KUKA KRL program: MyProgram_055().src

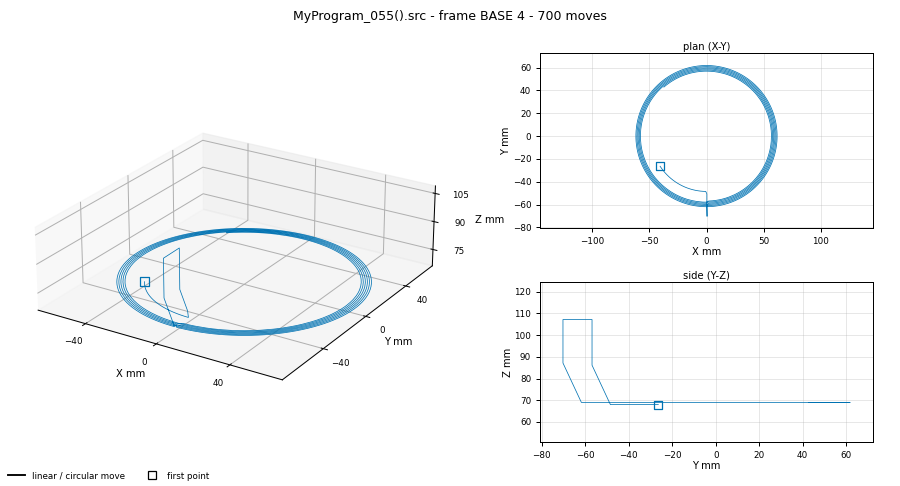
[picture p0: tool path of MyProgram_055().src in frame BASE 4, 700 of 700 moves have a stored position in this frame; points joined in program order, loops and branches not executed]
&ACCESS RVP
&REL 1
&PARAM TEMPLATE = C:\KRC\Roboter\Template\vorgabe
&PARAM EDITMASK = *
DEF MyProgram_055()
; ---- Setting reference (Base) ----
$BASE = BASE_DATA[4]

; --------------------------
; ---- Setting tool (TCP) ----
$TOOL = TOOL_DATA[3]
; --------------------------

$VEL.CP = VEL_APROX_PRINT
Startdeposition()
$VEL.CP = VEL_PRINT
LIN {X -40.6074,Y -26.4095,Z 68,A -152.5129,B 24.8688,C -2.6433,E1 24.8669,E2 236.0366} C_DIS
LIN {X -39.2547,Y -28.3812,Z 68,A -149.7049,B 24.8695,C -2.6361,E1 24.8714,E2 233.2321} C_DIS
LIN {X -37.8183,Y -30.2688,Z 68,A -146.8695,B 24.8701,C -2.63,E1 24.8763,E2 230.398} C_DIS
LIN {X -36.2912,Y -32.0839,Z 68,A -144.0489,B 24.8707,C -2.6239,E1 24.8814,E2 227.579} C_DIS
LIN {X -34.6958,Y -33.8024,Z 68,A -141.2485,B 24.8713,C -2.6184,E1 24.8868,E2 224.7796} C_DIS
LIN {X -32.9948,Y -35.4648,Z 68,A -138.4241,B 24.8718,C -2.6129,E1 24.8925,E2 221.9566} C_DIS
LIN {X -31.1918,Y -37.0607,Z 68,A -135.5745,B 24.8723,C -2.6076,E1 24.8986,E2 219.1087} C_DIS
LIN {X -29.3613,Y -38.5269,Z 68,A -132.7858,B 24.8728,C -2.6029,E1 24.9047,E2 216.3208} C_DIS
LIN {X -27.3998,Y -39.9459,Z 68,A -129.928,B 24.8733,C -2.5982,E1 24.9112,E2 213.4645} C_DIS
LIN {X -25.4106,Y -41.2399,Z 68,A -127.0866,B 24.8736,C -2.5945,E1 24.9179,E2 210.6229} C_DIS
LIN {X -23.4236,Y -42.3996,Z 68,A -124.332,B 24.8739,C -2.5914,E1 24.9246,E2 207.8677} C_DIS
LIN {X -21.2542,Y -43.5279,Z 68,A -121.4558,B 24.8743,C -2.5876,E1 24.9318,E2 204.9928} C_DIS
LIN {X -19.0978,Y -44.5162,Z 68,A -118.6602,B 24.8746,C -2.5844,E1 24.9389,E2 202.198} C_DIS
LIN {X -16.9499,Y -45.3772,Z 68,A -115.9012,B 24.8748,C -2.5823,E1 24.9461,E2 199.4383} C_DIS
LIN {X -14.6463,Y -46.1725,Z 68,A -113.0133,B 24.875,C -2.5801,E1 24.9538,E2 196.5502} C_DIS
LIN {X -12.4159,Y -46.8213,Z 68,A -110.2357,B 24.8751,C -2.5789,E1 24.9612,E2 193.7711} C_DIS
LIN {X -10.0365,Y -47.3887,Z 68,A -107.3856,B 24.8753,C -2.5768,E1 24.969,E2 190.9223} C_DIS
LIN {X -7.7033,Y -47.8234,Z 68,A -104.5763,B 24.8754,C -2.576,E1 24.9767,E2 188.1123} C_DIS
LIN {X -5.3374,Y -48.145,Z 68,A -101.7511,B 24.8754,C -2.5755,E1 24.9846,E2 185.2861} C_DIS
LIN {X -3.0451,Y -48.3437,Z 68,A -98.9821,B 24.8754,C -2.5763,E1 24.9923,E2 182.5142} C_DIS
LIN {X -0.6737,Y -48.4348,Z 68,A -96.2003,B 24.8754,C -2.5763,E1 25,E2 179.732} C_DIS
LIN {X -0.6737,Y -48.4348,Z 68,A -96.2003,B 24.8754,C -2.5763,E1 25,E2 179.732} C_DIS
Enddeposition()
LIN {X 0.3038,Y -50.5495,Z 72.5315,A -96.1445,B 24.8777,C -2.5529,E1 25,E2 179.732} C_DIS
LIN {X 0.2933,Y -56.8888,Z 86.1262,A -96.1143,B 24.8789,C -2.5402,E1 25,E2 179.732} C_DIS
LIN {X 0.2933,Y -56.8888,Z 107.1262,A -96.4674,B 24.8642,C -2.6887,E1 25,E2 179.732} C_DIS
LIN {X 0.4779,Y -70.2594,Z 107.1262,A -95.1787,B 24.8844,C -2.4821,E1 25.0023,E2 178.9343} C_DIS
LIN {X 0.4779,Y -70.2594,Z 87.1262,A -94.8425,B 24.8972,C -2.3406,E1 25.0023,E2 178.9343} C_DIS
LIN {X 0.4001,Y -63.9206,Z 73.5315,A -94.8701,B 24.8962,C -2.3523,E1 25.0023,E2 178.9343} C_DIS
LIN {X 0.3742,Y -61.8077,Z 69,A -94.8808,B 24.8958,C -2.3568,E1 25.0023,E2 178.9343} C_DIS
Startdeposition()
$VEL.CP = VEL_PRINT
LIN {X -1.5169,Y -61.7936,Z 69,A -97.6403,B 24.8977,C -2.3344,E1 24.9944,E2 181.747} C_DIS
LIN {X -4.5472,Y -61.6448,Z 69,A -100.4525,B 24.8977,C -2.3344,E1 24.9866,E2 184.5603} C_DIS
LIN {X -7.5665,Y -61.3474,Z 69,A -103.2657,B 24.8977,C -2.3346,E1 24.9788,E2 187.3745} C_DIS
LIN {X -10.5675,Y -60.9022,Z 69,A -106.0799,B 24.8977,C -2.3354,E1 24.971,E2 190.1896} C_DIS
LIN {X -13.5431,Y -60.3104,Z 69,A -108.8951,B 24.8976,C -2.3365,E1 24.9633,E2 193.0055} C_DIS
LIN {X -16.4861,Y -59.5732,Z 69,A -111.7113,B 24.8974,C -2.3381,E1 24.9557,E2 195.8221} C_DIS
LIN {X -19.3894,Y -58.6925,Z 69,A -114.5285,B 24.8973,C -2.34,E1 24.9482,E2 198.6396} C_DIS
LIN {X -22.2459,Y -57.6704,Z 69,A -117.3466,B 24.897,C -2.3424,E1 24.9408,E2 201.4578} C_DIS
LIN {X -25.0489,Y -56.5094,Z 69,A -120.1657,B 24.8968,C -2.3452,E1 24.9336,E2 204.2769} C_DIS
LIN {X -27.7915,Y -55.2122,Z 69,A -122.9858,B 24.8965,C -2.3484,E1 24.9265,E2 207.0968} C_DIS
LIN {X -30.4671,Y -53.782,Z 69,A -125.8067,B 24.8962,C -2.3519,E1 24.9196,E2 209.9173} C_DIS
LIN {X -33.0694,Y -52.2223,Z 69,A -128.6284,B 24.8959,C -2.3558,E1 24.9129,E2 212.7385} C_DIS
LIN {X -35.592,Y -50.5368,Z 69,A -131.4511,B 24.8955,C -2.3601,E1 24.9064,E2 215.5605} C_DIS
LIN {X -38.0289,Y -48.7295,Z 69,A -134.2747,B 24.8951,C -2.3648,E1 24.9001,E2 218.3832} C_DIS
LIN {X -40.3741,Y -46.8048,Z 69,A -137.0991,B 24.8946,C -2.3698,E1 24.8941,E2 221.2065} C_DIS
LIN {X -42.6125,Y -44.7764,Z 69,A -139.915,B 24.8942,C -2.375,E1 24.8883,E2 224.0214} C_DIS
LIN {X -44.7673,Y -42.6221,Z 69,A -142.7502,B 24.8936,C -2.3807,E1 24.8828,E2 226.8551} C_DIS
LIN {X -46.8048,Y -40.3741,Z 69,A -145.5768,B 24.8931,C -2.3867,E1 24.8776,E2 229.6802} C_DIS
LIN {X -48.7295,Y -38.0289,Z 69,A -148.4042,B 24.8925,C -2.393,E1 24.8727,E2 232.5058} C_DIS
LIN {X -50.5368,Y -35.592,Z 69,A -151.2322,B 24.892,C -2.3995,E1 24.868,E2 235.332} C_DIS
LIN {X -52.2223,Y -33.0694,Z 69,A -154.0608,B 24.8913,C -2.4063,E1 24.8637,E2 238.1586} C_DIS
LIN {X -53.782,Y -30.4671,Z 69,A -156.8901,B 24.8907,C -2.4133,E1 24.8597,E2 240.9858} C_DIS
LIN {X -55.2122,Y -27.7915,Z 69,A -159.7199,B 24.89,C -2.4206,E1 24.8561,E2 243.8133} C_DIS
LIN {X -56.5094,Y -25.0489,Z 69,A -162.5501,B 24.8894,C -2.4281,E1 24.8528,E2 246.6411} C_DIS
LIN {X -57.6704,Y -22.2459,Z 69,A -165.3808,B 24.8887,C -2.4357,E1 24.8499,E2 249.4694} C_DIS
LIN {X -58.6925,Y -19.3894,Z 69,A -168.212,B 24.8879,C -2.4436,E1 24.8473,E2 252.298} C_DIS
LIN {X -59.5732,Y -16.4861,Z 69,A -171.0435,B 24.8872,C -2.4516,E1 24.8451,E2 255.1266} C_DIS
LIN {X -60.3104,Y -13.5431,Z 69,A -173.8753,B 24.8864,C -2.4597,E1 24.8433,E2 257.9557} C_DIS
LIN {X -60.9022,Y -10.5675,Z 69,A -176.7075,B 24.8857,C -2.468,E1 24.8418,E2 260.7849} C_DIS
LIN {X -61.3474,Y -7.5665,Z 69,A -179.5398,B 24.8849,C -2.4763,E1 24.8408,E2 263.6142} C_DIS
LIN {X -61.6448,Y -4.5472,Z 69,A 177.6277,B 24.8841,C -2.4847,E1 24.8401,E2 266.4436} C_DIS
LIN {X -61.7936,Y -1.5169,Z 69,A 174.8866,B 24.8832,C -2.4949,E1 24.8398,E2 269.177} C_DIS
LIN {X -61.7936,Y 1.5169,Z 69,A 171.9622,B 24.8825,C -2.5017,E1 24.8398,E2 272.1025} C_DIS
LIN {X -61.6448,Y 4.5472,Z 69,A 169.1296,B 24.8817,C -2.5102,E1 24.8404,E2 274.9319} C_DIS
LIN {X -61.3474,Y 7.5665,Z 69,A 166.2969,B 24.8809,C -2.5188,E1 24.8412,E2 277.7612} C_DIS
LIN {X -60.9022,Y 10.5675,Z 69,A 163.4642,B 24.8801,C -2.5272,E1 24.8425,E2 280.5904} C_DIS
LIN {X -60.3104,Y 13.5431,Z 69,A 160.6317,B 24.8793,C -2.5357,E1 24.8441,E2 283.4195} C_DIS
LIN {X -59.5732,Y 16.4861,Z 69,A 157.7993,B 24.8785,C -2.544,E1 24.8461,E2 286.2484} C_DIS
LIN {X -58.6925,Y 19.3894,Z 69,A 154.9672,B 24.8777,C -2.5523,E1 24.8485,E2 289.077} C_DIS
LIN {X -57.6704,Y 22.2459,Z 69,A 152.1353,B 24.8769,C -2.5605,E1 24.8513,E2 291.9053} C_DIS
LIN {X -56.5094,Y 25.0489,Z 69,A 149.3037,B 24.8761,C -2.5685,E1 24.8544,E2 294.7334} C_DIS
LIN {X -55.2122,Y 27.7915,Z 69,A 146.4725,B 24.8754,C -2.5763,E1 24.8578,E2 297.5612} C_DIS
LIN {X -53.782,Y 30.4671,Z 69,A 143.6416,B 24.8746,C -2.584,E1 24.8616,E2 300.3885} C_DIS
LIN {X -52.2223,Y 33.0694,Z 69,A 140.8113,B 24.8739,C -2.5916,E1 24.8658,E2 303.2154} C_DIS
LIN {X -50.5368,Y 35.592,Z 69,A 137.9814,B 24.8732,C -2.5989,E1 24.8702,E2 306.0419} C_DIS
LIN {X -48.7295,Y 38.0289,Z 69,A 135.1522,B 24.8725,C -2.606,E1 24.875,E2 308.8677} C_DIS
LIN {X -46.8048,Y 40.3741,Z 69,A 132.3234,B 24.8718,C -2.6128,E1 24.8801,E2 311.6931} C_DIS
LIN {X -44.7673,Y 42.6221,Z 69,A 129.4952,B 24.8712,C -2.6194,E1 24.8855,E2 314.518} C_DIS
LIN {X -42.6221,Y 44.7673,Z 69,A 126.6678,B 24.8706,C -2.6257,E1 24.8911,E2 317.3422} C_DIS
LIN {X -40.3741,Y 46.8048,Z 69,A 123.8408,B 24.87,C -2.6317,E1 24.897,E2 320.166} C_DIS
LIN {X -38.0289,Y 48.7295,Z 69,A 121.0148,B 24.8694,C -2.6374,E1 24.9032,E2 322.9889} C_DIS
LIN {X -35.592,Y 50.5368,Z 69,A 118.1895,B 24.8689,C -2.6428,E1 24.9095,E2 325.8113} C_DIS
LIN {X -33.0694,Y 52.2223,Z 69,A 115.365,B 24.8683,C -2.6479,E1 24.9161,E2 328.6328} C_DIS
LIN {X -30.4671,Y 53.782,Z 69,A 112.5412,B 24.8679,C -2.6526,E1 24.9229,E2 331.4539} C_DIS
LIN {X -27.8247,Y 55.1952,Z 69,A 109.7441,B 24.8675,C -2.6567,E1 24.9299,E2 334.2487} C_DIS
LIN {X -25.0489,Y 56.5094,Z 69,A 106.8964,B 24.867,C -2.661,E1 24.9371,E2 337.0934} C_DIS
LIN {X -22.2459,Y 57.6704,Z 69,A 104.0752,B 24.8667,C -2.6646,E1 24.9444,E2 339.9121} C_DIS
LIN {X -19.3894,Y 58.6925,Z 69,A 101.2549,B 24.8663,C -2.6678,E1 24.9518,E2 342.7301} C_DIS
LIN {X -16.4861,Y 59.5732,Z 69,A 98.4357,B 24.8661,C -2.6707,E1 24.9594,E2 345.5471} C_DIS
LIN {X -13.5431,Y 60.3104,Z 69,A 95.6173,B 24.8658,C -2.6731,E1 24.967,E2 348.3634} C_DIS
LIN {X -10.5675,Y 60.9022,Z 69,A 92.7999,B 24.8656,C -2.6752,E1 24.9748,E2 351.179} C_DIS
LIN {X -7.6019,Y 61.3428,Z 69,A 90.0082,B 24.8655,C -2.6767,E1 24.9825,E2 353.9694} C_DIS
LIN {X -4.5472,Y 61.6448,Z 69,A 87.168,B 24.8653,C -2.6781,E1 24.9904,E2 356.8075} C_DIS
LIN {X -1.5169,Y 61.7936,Z 69,A 84.3535,B 24.8653,C -2.6789,E1 24.9982,E2 359.6205} C_DIS
LIN {X 1.5169,Y 61.7936,Z 69,A 81.54,B 24.8652,C -2.6793,E1 25.0061,E2 362.4328} C_DIS
LIN {X 4.5472,Y 61.6448,Z 69,A 78.7275,B 24.8652,C -2.6793,E1 25.0139,E2 365.244} C_DIS
LIN {X 7.5665,Y 61.3474,Z 69,A 75.9161,B 24.8652,C -2.6789,E1 25.0217,E2 368.0545} C_DIS
LIN {X 10.5675,Y 60.9022,Z 69,A 73.1055,B 24.8653,C -2.6781,E1 25.0295,E2 370.8643} C_DIS
LIN {X 13.5431,Y 60.3104,Z 69,A 70.296,B 24.8654,C -2.6769,E1 25.0371,E2 373.6732} C_DIS
LIN {X 16.4861,Y 59.5732,Z 69,A 67.4874,B 24.8656,C -2.6752,E1 25.0447,E2 376.4812} C_DIS
LIN {X 19.3894,Y 58.6925,Z 69,A 64.6798,B 24.8658,C -2.6732,E1 25.0522,E2 379.2886} C_DIS
LIN {X 22.2459,Y 57.6704,Z 69,A 61.8732,B 24.8661,C -2.6707,E1 25.0596,E2 382.0951} C_DIS
LIN {X 25.0489,Y 56.5094,Z 69,A 59.0674,B 24.8663,C -2.6679,E1 25.0668,E2 384.9009} C_DIS
LIN {X 27.7915,Y 55.2122,Z 69,A 56.2625,B 24.8667,C -2.6646,E1 25.0738,E2 387.706} C_DIS
LIN {X 30.4671,Y 53.782,Z 69,A 53.4587,B 24.867,C -2.661,E1 25.0807,E2 390.5102} C_DIS
LIN {X 33.0694,Y 52.2223,Z 69,A 50.6555,B 24.8674,C -2.6571,E1 25.0873,E2 393.314} C_DIS
LIN {X 35.592,Y 50.5368,Z 69,A 47.8533,B 24.8679,C -2.6528,E1 25.0938,E2 396.1169} C_DIS
LIN {X 38.0289,Y 48.7295,Z 69,A 45.0519,B 24.8683,C -2.6481,E1 25.1,E2 398.9192} C_DIS
LIN {X 40.3741,Y 46.8048,Z 69,A 42.2512,B 24.8688,C -2.6431,E1 25.106,E2 401.7209} C_DIS
LIN {X 42.6221,Y 44.7673,Z 69,A 39.4515,B 24.8694,C -2.6377,E1 25.1117,E2 404.5219} C_DIS
LIN {X 44.7673,Y 42.6221,Z 69,A 36.6525,B 24.8699,C -2.6321,E1 25.1172,E2 407.3223} C_DIS
LIN {X 46.8048,Y 40.3741,Z 69,A 33.8542,B 24.8705,C -2.6261,E1 25.1224,E2 410.1222} C_DIS
LIN {X 48.7295,Y 38.0289,Z 69,A 31.0563,B 24.8711,C -2.6199,E1 25.1273,E2 412.9217} C_DIS
LIN {X 50.5368,Y 35.592,Z 69,A 28.2593,B 24.8718,C -2.6134,E1 25.1318,E2 415.7205} C_DIS
LIN {X 52.2223,Y 33.0694,Z 69,A 25.4629,B 24.8724,C -2.6067,E1 25.1361,E2 418.5189} C_DIS
LIN {X 53.782,Y 30.4671,Z 69,A 22.667,B 24.8731,C -2.5997,E1 25.14,E2 421.3169} C_DIS
LIN {X 55.2122,Y 27.7915,Z 69,A 19.8717,B 24.8738,C -2.5925,E1 25.1436,E2 424.1145} C_DIS
LIN {X 56.5094,Y 25.0489,Z 69,A 17.0768,B 24.8745,C -2.5851,E1 25.1469,E2 426.9117} C_DIS
LIN {X 57.6704,Y 22.2459,Z 69,A 14.2823,B 24.8753,C -2.5775,E1 25.1498,E2 429.7087} C_DIS
LIN {X 58.6925,Y 19.3894,Z 69,A 11.4883,B 24.876,C -2.5697,E1 25.1523,E2 432.5054} C_DIS
LIN {X 59.5732,Y 16.4861,Z 69,A 8.6946,B 24.8768,C -2.5618,E1 25.1545,E2 435.3019} C_DIS
LIN {X 60.3104,Y 13.5431,Z 69,A 5.9012,B 24.8776,C -2.5537,E1 25.1563,E2 438.098} C_DIS
LIN {X 60.9022,Y 10.5675,Z 69,A 3.1081,B 24.8784,C -2.5456,E1 25.1578,E2 440.8941} C_DIS
LIN {X 61.3474,Y 7.5665,Z 69,A 0.3152,B 24.8791,C -2.5373,E1 25.1588,E2 443.6901} C_DIS
LIN {X 61.6448,Y 4.5472,Z 69,A -2.4776,B 24.8799,C -2.529,E1 25.1595,E2 446.4859} C_DIS
LIN {X 61.7936,Y 1.5169,Z 69,A -5.18,B 24.8805,C -2.5229,E1 25.1598,E2 449.1868} C_DIS
LIN {X 61.7936,Y -1.5169,Z 69,A -8.0628,B 24.8815,C -2.5122,E1 25.1597,E2 452.0775} C_DIS
LIN {X 61.6448,Y -4.5472,Z 69,A -10.8552,B 24.8823,C -2.5038,E1 25.1592,E2 454.8732} C_DIS
LIN {X 61.3474,Y -7.5665,Z 69,A -13.6477,B 24.8831,C -2.4954,E1 25.1583,E2 457.6691} C_DIS
LIN {X 60.9022,Y -10.5675,Z 69,A -16.4402,B 24.8839,C -2.487,E1 25.1571,E2 460.4651} C_DIS
LIN {X 60.3104,Y -13.5431,Z 69,A -19.2329,B 24.8847,C -2.4787,E1 25.1555,E2 463.2612} C_DIS
LIN {X 59.5732,Y -16.4861,Z 69,A -22.0257,B 24.8855,C -2.4704,E1 25.1535,E2 466.0575} C_DIS
LIN {X 58.6925,Y -19.3894,Z 69,A -24.8188,B 24.8862,C -2.4622,E1 25.1511,E2 468.854} C_DIS
LIN {X 57.6704,Y -22.2459,Z 69,A -27.612,B 24.887,C -2.4542,E1 25.1484,E2 471.6507} C_DIS
LIN {X 56.5094,Y -25.0489,Z 69,A -30.4057,B 24.8877,C -2.4462,E1 25.1454,E2 474.4479} C_DIS
LIN {X 55.2122,Y -27.7915,Z 69,A -33.1997,B 24.8884,C -2.4384,E1 25.1419,E2 477.2454} C_DIS
LIN {X 53.782,Y -30.4671,Z 69,A -35.994,B 24.8891,C -2.4307,E1 25.1382,E2 480.0432} C_DIS
LIN {X 52.2223,Y -33.0694,Z 69,A -38.7886,B 24.8898,C -2.4233,E1 25.1341,E2 482.8413} C_DIS
LIN {X 50.5368,Y -35.592,Z 69,A -41.5839,B 24.8905,C -2.416,E1 25.1296,E2 485.6399} C_DIS
LIN {X 48.7295,Y -38.0289,Z 69,A -44.3797,B 24.8911,C -2.4089,E1 25.1249,E2 488.4391} C_DIS
LIN {X 46.8048,Y -40.3741,Z 69,A -47.1759,B 24.8917,C -2.4021,E1 25.1199,E2 491.2387} C_DIS
LIN {X 44.7673,Y -42.6221,Z 69,A -49.9729,B 24.8923,C -2.3955,E1 25.1146,E2 494.039} C_DIS
LIN {X 42.6221,Y -44.7673,Z 69,A -52.7703,B 24.8929,C -2.3892,E1 25.109,E2 496.8396} C_DIS
LIN {X 40.3741,Y -46.8048,Z 69,A -55.5685,B 24.8934,C -2.3832,E1 25.1031,E2 499.641} C_DIS
LIN {X 38.0289,Y -48.7295,Z 69,A -58.3673,B 24.8939,C -2.3775,E1 25.097,E2 502.4429} C_DIS
LIN {X 35.592,Y -50.5368,Z 69,A -61.1669,B 24.8944,C -2.372,E1 25.0907,E2 505.2455} C_DIS
LIN {X 33.0694,Y -52.2223,Z 69,A -63.9673,B 24.8949,C -2.3669,E1 25.0841,E2 508.0487} C_DIS
LIN {X 30.4671,Y -53.782,Z 69,A -66.7685,B 24.8953,C -2.3622,E1 25.0773,E2 510.8528} C_DIS
LIN {X 27.7915,Y -55.2122,Z 69,A -69.5705,B 24.8957,C -2.3577,E1 25.0704,E2 513.6574} C_DIS
LIN {X 25.0489,Y -56.5094,Z 69,A -72.3733,B 24.8961,C -2.3537,E1 25.0633,E2 516.4628} C_DIS
LIN {X 22.2459,Y -57.6704,Z 69,A -75.177,B 24.8964,C -2.35,E1 25.056,E2 519.269} C_DIS
LIN {X 19.3894,Y -58.6925,Z 69,A -77.9817,B 24.8967,C -2.3466,E1 25.0486,E2 522.076} C_DIS
LIN {X 16.4861,Y -59.5732,Z 69,A -80.7871,B 24.8969,C -2.3437,E1 25.0411,E2 524.8836} C_DIS
LIN {X 13.5431,Y -60.3104,Z 69,A -83.5936,B 24.8972,C -2.3411,E1 25.0334,E2 527.6921} C_DIS
LIN {X 10.5675,Y -60.9022,Z 69,A -86.401,B 24.8973,C -2.339,E1 25.0257,E2 530.5015} C_DIS
LIN {X 7.5665,Y -61.3474,Z 69,A -89.2093,B 24.8975,C -2.3372,E1 25.0179,E2 533.3116} C_DIS
LIN {X 4.5472,Y -61.6448,Z 69,A -92.0187,B 24.8976,C -2.3359,E1 25.0101,E2 536.1226} C_DIS
LIN {X 1.5169,Y -61.7936,Z 69,A -94.829,B 24.8977,C -2.335,E1 25.0023,E2 538.9343} C_DIS
LIN {X 1.5169,Y -61.7936,Z 69,A -94.829,B 24.8977,C -2.335,E1 25.0023,E2 538.9343} C_DIS
Enddeposition()
LIN {X 0.3699,Y -60.8218,Z 69,A -95.3511,B 24.8952,C -2.3637,E1 25.001,E2 539.3882} C_DIS
Startdeposition()
$VEL.CP = VEL_PRINT
LIN {X 3.5241,Y -60.721,Z 69,A -91.7282,B 24.8938,C -2.3788,E1 25.0112,E2 535.7302} C_DIS
LIN {X 6.9367,Y -60.4263,Z 69,A -88.4115,B 24.8935,C -2.3825,E1 25.0205,E2 532.4068} C_DIS
LIN {X 9.7316,Y -60.0402,Z 69,A -84.8923,B 24.8916,C -2.4038,E1 25.0303,E2 528.8406} C_DIS
LIN {X 13.0357,Y -59.4097,Z 69,A -82.7107,B 24.8933,C -2.3843,E1 25.0361,E2 526.7081} C_DIS
LIN {X 15.5224,Y -58.81,Z 69,A -80.1105,B 24.8927,C -2.391,E1 25.0432,E2 524.0959} C_DIS
LIN {X 17.6784,Y -58.1982,Z 69,A -78.3032,B 24.8931,C -2.3864,E1 25.048,E2 522.3025} C_DIS
LIN {X 20.9532,Y -57.1,Z 69,A -74.8965,B 24.8925,C -2.394,E1 25.057,E2 518.8847} C_DIS
LIN {X 23.4984,Y -56.1006,Z 69,A -72.2344,B 24.8919,C -2.3996,E1 25.0639,E2 516.2154} C_DIS
LIN {X 26.0446,Y -54.9656,Z 69,A -68.804,B 24.8899,C -2.4224,E1 25.0727,E2 512.7398} C_DIS
LIN {X 29.0105,Y -53.4586,Z 69,A -66.3744,B 24.8909,C -2.4112,E1 25.0786,E2 510.3437} C_DIS
LIN {X 31.8828,Y -51.798,Z 69,A -63.3879,B 24.8907,C -2.4135,E1 25.0857,E2 507.3608} C_DIS
LIN {X 34.4186,Y -50.1491,Z 69,A -60.7942,B 24.8907,C -2.4131,E1 25.0917,E2 504.7769} C_DIS
LIN {X 37.3365,Y -48.0155,Z 69,A -57.1659,B 24.8896,C -2.4254,E1 25.0999,E2 501.1324} C_DIS
LIN {X 39.6383,Y -46.1336,Z 69,A -54.7199,B 24.8898,C -2.4231,E1 25.1051,E2 498.7012} C_DIS
LIN {X 41.8601,Y -44.1275,Z 69,A -51.5668,B 24.8885,C -2.4376,E1 25.1116,E2 495.5267} C_DIS
LIN {X 44.7982,Y -41.1407,Z 69,A -47.6443,B 24.8877,C -2.4466,E1 25.1192,E2 491.5998} C_DIS
LIN {X 46.9752,Y -38.6376,Z 69,A -44.2528,B 24.8863,C -2.461,E1 25.1254,E2 488.1896} C_DIS
LIN {X 49.0255,Y -35.9992,Z 69,A -41.6748,B 24.8868,C -2.4556,E1 25.1297,E2 485.6369} C_DIS
LIN {X 50.7232,Y -33.565,Z 69,A -38.4521,B 24.8852,C -2.4736,E1 25.1348,E2 482.3874} C_DIS
LIN {X 52.2264,Y -31.1755,Z 69,A -35.773,B 24.8844,C -2.4816,E1 25.1386,E2 479.7031} C_DIS
LIN {X 53.8881,Y -28.2053,Z 69,A -32.8097,B 24.8841,C -2.4849,E1 25.1426,E2 476.7475} C_DIS
LIN {X 55.2151,Y -25.5099,Z 69,A -30.0221,B 24.8834,C -2.4922,E1 25.1459,E2 473.9577} C_DIS
LIN {X 56.1602,Y -23.3571,Z 69,A -27.557,B 24.8822,C -2.505,E1 25.1486,E2 471.476} C_DIS
LIN {X 57.3545,Y -20.2464,Z 69,A -24.8024,B 24.8822,C -2.505,E1 25.1513,E2 468.7365} C_DIS
LIN {X 58.0728,Y -18.083,Z 69,A -22.7658,B 24.8818,C -2.5089,E1 25.153,E2 466.7024} C_DIS
LIN {X 58.8136,Y -15.5078,Z 69,A -20.0069,B 24.8806,C -2.5225,E1 25.155,E2 463.9271} C_DIS
LIN {X 59.6377,Y -11.9522,Z 69,A -16.6322,B 24.8797,C -2.5317,E1 25.1571,E2 460.5503} C_DIS
LIN {X 60.0812,Y -9.4722,Z 69,A -13.8457,B 24.878,C -2.5495,E1 25.1583,E2 457.7383} C_DIS
LIN {X 60.5662,Y -5.5828,Z 69,A -10.6448,B 24.878,C -2.5489,E1 25.1593,E2 454.5575} C_DIS
LIN {X 60.7566,Y -2.8512,Z 69,A -8.1375,B 24.8774,C -2.5553,E1 25.1597,E2 452.05} C_DIS
LIN {X 60.8244,Y -0.2246,Z 69,A -5.502,B 24.8763,C -2.5671,E1 25.1597,E2 449.4025} C_DIS
LIN {X 60.7088,Y 3.7418,Z 69,A -1.8226,B 24.8753,C -2.5774,E1 25.1593,E2 445.7205} C_DIS
LIN {X 60.3426,Y 7.6319,Z 69,A 1.9824,B 24.8739,C -2.5919,E1 25.1582,E2 441.9037} C_DIS
LIN {X 59.8211,Y 10.9965,Z 69,A 5.4528,B 24.8723,C -2.6083,E1 25.1565,E2 438.4149} C_DIS
LIN {X 58.6681,Y 16.0475,Z 69,A 9.7585,B 24.8723,C -2.6088,E1 25.1536,E2 434.1328} C_DIS
LIN {X 57.8754,Y 18.705,Z 69,A 12.3693,B 24.8715,C -2.6165,E1 25.1515,E2 431.5186} C_DIS
LIN {X 56.9734,Y 21.2964,Z 69,A 14.8842,B 24.8709,C -2.6223,E1 25.1491,E2 429.0041} C_DIS
LIN {X 55.9024,Y 23.9686,Z 69,A 17.7553,B 24.8697,C -2.6339,E1 25.146,E2 426.1216} C_DIS
LIN {X 54.968,Y 26.0397,Z 69,A 19.8777,B 24.8692,C -2.6393,E1 25.1435,E2 423.9977} C_DIS
LIN {X 53.6349,Y 28.6855,Z 69,A 22.5302,B 24.8688,C -2.6436,E1 25.1401,E2 421.3492} C_DIS
LIN {X 52.3266,Y 31.0059,Z 69,A 25.1098,B 24.868,C -2.6519,E1 25.1365,E2 418.7633} C_DIS
LIN {X 51.0461,Y 33.0727,Z 69,A 27.3319,B 24.8675,C -2.6561,E1 25.1331,E2 416.5424} C_DIS
LIN {X 49.5259,Y 35.3075,Z 69,A 29.8988,B 24.8668,C -2.6628,E1 25.129,E2 413.972} C_DIS
LIN {X 47.6836,Y 37.7586,Z 69,A 32.4782,B 24.8668,C -2.6624,E1 25.1246,E2 411.406} C_DIS
LIN {X 44.7969,Y 41.1421,Z 69,A 37.0286,B 24.8651,C -2.6803,E1 25.1163,E2 406.8337} C_DIS
LIN {X 42.4394,Y 43.5711,Z 69,A 39.7141,B 24.8656,C -2.6752,E1 25.111,E2 404.1717} C_DIS
LIN {X 39.5796,Y 46.1836,Z 69,A 43.7208,B 24.864,C -2.6906,E1 25.1027,E2 400.1445} C_DIS
LIN {X 37.4821,Y 47.9022,Z 69,A 46.1859,B 24.8638,C -2.6932,E1 25.0973,E2 397.6825} C_DIS
LIN {X 35.4881,Y 49.3971,Z 69,A 48.479,B 24.8635,C -2.6959,E1 25.0921,E2 395.3911} C_DIS
LIN {X 33.2095,Y 50.9575,Z 69,A 50.9932,B 24.8633,C -2.6981,E1 25.0863,E2 392.8802} C_DIS
LIN {X 31.29,Y 52.1582,Z 69,A 53.1478,B 24.8629,C -2.7017,E1 25.0812,E2 390.7237} C_DIS
LIN {X 29.1742,Y 53.3699,Z 69,A 55.6356,B 24.8622,C -2.7092,E1 25.0751,E2 388.2256} C_DIS
LIN {X 26.4475,Y 54.7721,Z 69,A 58.483,B 24.8619,C -2.7118,E1 25.068,E2 385.3796} C_DIS
LIN {X 23.9448,Y 55.9125,Z 69,A 61.1419,B 24.8614,C -2.7162,E1 25.0612,E2 382.7169} C_DIS
LIN {X 21.3004,Y 56.9719,Z 69,A 63.7978,B 24.8612,C -2.7181,E1 25.0542,E2 380.0621} C_DIS
LIN {X 18.5844,Y 57.9144,Z 69,A 66.505,B 24.861,C -2.7203,E1 25.0471,E2 377.3549} C_DIS
LIN {X 16.1062,Y 58.6523,Z 69,A 69.0598,B 24.8606,C -2.7245,E1 25.0402,E2 374.7944} C_DIS
LIN {X 12.5567,Y 59.5137,Z 69,A 72.275,B 24.8609,C -2.7213,E1 25.0315,E2 371.591} C_DIS
LIN {X 9.9654,Y 60.0011,Z 69,A 74.4475,B 24.8615,C -2.7156,E1 25.0255,E2 369.4347} C_DIS
LIN {X 7.7997,Y 60.3208,Z 69,A 78.057,B 24.858,C -2.7494,E1 25.0153,E2 365.7477} C_DIS
LIN {X 3.6725,Y 60.7128,Z 69,A 80.3983,B 24.8615,C -2.716,E1 25.009,E2 363.4869} C_DIS
LIN {X -0.0244,Y 60.824,Z 69,A 84.239,B 24.8607,C -2.723,E1 24.9983,E2 359.6301} C_DIS
LIN {X -2.9809,Y 60.751,Z 69,A 86.9887,B 24.8609,C -2.7214,E1 24.9906,E2 356.8837} C_DIS
LIN {X -5.8016,Y 60.546,Z 69,A 89.7033,B 24.8609,C -2.7213,E1 24.983,E2 354.1683} C_DIS
LIN {X -10.4137,Y 59.9255,Z 69,A 94.0806,B 24.8612,C -2.7182,E1 24.971,E2 349.7945} C_DIS
LIN {X -13.7016,Y 59.2596,Z 69,A 97.2928,B 24.8614,C -2.7166,E1 24.9622,E2 346.5823} C_DIS
LIN {X -16.4479,Y 58.557,Z 69,A 99.9665,B 24.8617,C -2.714,E1 24.955,E2 343.9107} C_DIS
LIN {X -19.0418,Y 57.7663,Z 69,A 102.4277,B 24.8622,C -2.7092,E1 24.9485,E2 341.4566} C_DIS
LIN {X -23.2617,Y 56.1995,Z 69,A 106.3977,B 24.8633,C -2.6983,E1 24.9382,E2 337.5041} C_DIS
LIN {X -26.378,Y 54.8054,Z 69,A 109.7592,B 24.8635,C -2.6964,E1 24.9296,E2 334.139} C_DIS
LIN {X -27.9233,Y 54.0352,Z 69,A 112.467,B 24.8616,C -2.715,E1 24.9228,E2 331.3795} C_DIS
LIN {X -30.8335,Y 52.4285,Z 69,A 114.7128,B 24.8639,C -2.6922,E1 24.9175,E2 329.1814} C_DIS
LIN {X -33.2267,Y 50.9462,Z 69,A 117.3953,B 24.8643,C -2.6878,E1 24.9111,E2 326.5007} C_DIS
LIN {X -35.6247,Y 49.2996,Z 69,A 120.2042,B 24.8647,C -2.6837,E1 24.9047,E2 323.6919} C_DIS
LIN {X -38.0459,Y 47.4557,Z 69,A 123.3465,B 24.8648,C -2.683,E1 24.8978,E2 320.5398} C_DIS
LIN {X -41.0603,Y 44.872,Z 69,A 126.7217,B 24.8664,C -2.6677,E1 24.8908,E2 317.1877} C_DIS
LIN {X -43.1122,Y 42.9049,Z 69,A 129.5063,B 24.8668,C -2.6634,E1 24.8852,E2 314.4016} C_DIS
LIN {X -45.1474,Y 40.7579,Z 69,A 131.8856,B 24.8682,C -2.649,E1 24.8807,E2 312.0463} C_DIS
LIN {X -46.6661,Y 39.0096,Z 69,A 135.0862,B 24.8669,C -2.6625,E1 24.8749,E2 308.7988} C_DIS
LIN {X -49.2279,Y 35.7228,Z 69,A 138.4377,B 24.869,C -2.6414,E1 24.8693,E2 305.4817} C_DIS
LIN {X -50.7628,Y 33.5048,Z 69,A 141.0102,B 24.8696,C -2.6351,E1 24.8653,E2 302.9115} C_DIS
LIN {X -52.0957,Y 31.3931,Z 69,A 143.9984,B 24.8691,C -2.6403,E1 24.861,E2 299.8955} C_DIS
LIN {X -54.1446,Y 27.7093,Z 69,A 147.3916,B 24.8713,C -2.6182,E1 24.8565,E2 296.5371} C_DIS
LIN {X -55.184,Y 25.5767,Z 69,A 149.7296,B 24.8718,C -2.6135,E1 24.8538,E2 294.1975} C_DIS
LIN {X -56.4618,Y 22.619,Z 69,A 152.6761,B 24.8728,C -2.6028,E1 24.8506,E2 291.2603} C_DIS
LIN {X -57.4388,Y 20.0061,Z 69,A 155.3015,B 24.8736,C -2.5948,E1 24.8481,E2 288.6391} C_DIS
LIN {X -58.2751,Y 17.4201,Z 69,A 157.8501,B 24.8744,C -2.5868,E1 24.846,E2 286.0952} C_DIS
LIN {X -59.0128,Y 14.7319,Z 69,A 160.1902,B 24.8757,C -2.5735,E1 24.8444,E2 283.7732} C_DIS
LIN {X -59.433,Y 12.9288,Z 69,A 162.2542,B 24.8757,C -2.5738,E1 24.8431,E2 281.6962} C_DIS
LIN {X -59.964,Y 10.1871,Z 69,A 164.8902,B 24.8764,C -2.5656,E1 24.8418,E2 279.0641} C_DIS
LIN {X -60.3844,Y 7.2944,Z 69,A 167.7265,B 24.8771,C -2.5584,E1 24.8407,E2 276.2282} C_DIS
LIN {X -60.6651,Y 4.379,Z 69,A 170.6353,B 24.8777,C -2.5524,E1 24.84,E2 273.3162} C_DIS
LIN {X -60.7919,Y 1.9468,Z 69,A 172.5622,B 24.879,C -2.5386,E1 24.8398,E2 271.4109} C_DIS
LIN {X -60.8219,Y -0.493,Z 69,A 175.2013,B 24.8791,C -2.5374,E1 24.8398,E2 268.7585} C_DIS
LIN {X -60.7323,Y -3.3196,Z 69,A 177.8663,B 24.8799,C -2.5291,E1 24.8401,E2 266.0974} C_DIS
LIN {X -60.5142,Y -6.1249,Z 69,A -179.6063,B 24.8809,C -2.5186,E1 24.8408,E2 263.5799} C_DIS
LIN {X -60.1684,Y -8.9064,Z 69,A -176.772,B 24.8814,C -2.5139,E1 24.8419,E2 260.7399} C_DIS
LIN {X -59.6262,Y -12.0083,Z 69,A -173.9619,B 24.8825,C -2.502,E1 24.8433,E2 257.9417} C_DIS
LIN {X -59.0014,Y -14.7785,Z 69,A -171.3606,B 24.8834,C -2.4926,E1 24.845,E2 255.3476} C_DIS
LIN {X -58.5565,Y -16.4495,Z 69,A -169.5667,B 24.8836,C -2.4908,E1 24.8463,E2 253.5477} C_DIS
LIN {X -57.7201,Y -19.1807,Z 69,A -166.836,B 24.8842,C -2.4836,E1 24.8486,E2 250.8185} C_DIS
LIN {X -56.7436,Y -21.9028,Z 69,A -164.0819,B 24.8849,C -2.4763,E1 24.8513,E2 248.0663} C_DIS
LIN {X -54.6571,Y -26.6865,Z 69,A -158.7948,B 24.8855,C -2.4695,E1 24.8574,E2 242.7665} C_DIS
LIN {X -52.9066,Y -30.0074,Z 69,A -155.8669,B 24.8875,C -2.4487,E1 24.8613,E2 239.8728} C_DIS
LIN {X -51.7465,Y -31.9661,Z 69,A -153.4161,B 24.8875,C -2.4489,E1 24.8648,E2 237.409} C_DIS
LIN {X -50.2012,Y -34.3418,Z 69,A -150.7503,B 24.8881,C -2.4421,E1 24.869,E2 234.746} C_DIS
LIN {X -48.6003,Y -36.5712,Z 69,A -148.1528,B 24.8886,C -2.4361,E1 24.8733,E2 232.1502} C_DIS
LIN {X -46.7849,Y -38.8665,Z 69,A -145.4654,B 24.8893,C -2.4284,E1 24.878,E2 229.4687} C_DIS
LIN {X -45.1324,Y -40.7747,Z 69,A -142.9432,B 24.8896,C -2.4259,E1 24.8827,E2 226.9412} C_DIS
LIN {X -43.0487,Y -42.9691,Z 69,A -140.1657,B 24.8902,C -2.4185,E1 24.888,E2 224.1695} C_DIS
LIN {X -41.0534,Y -44.8783,Z 69,A -137.4786,B 24.8905,C -2.415,E1 24.8935,E2 221.4797} C_DIS
LIN {X -38.8702,Y -46.7818,Z 69,A -134.7466,B 24.891,C -2.4099,E1 24.8993,E2 218.7491} C_DIS
LIN {X -36.6016,Y -48.5774,Z 69,A -132.1771,B 24.8917,C -2.4021,E1 24.905,E2 216.189} C_DIS
LIN {X -34.4272,Y -50.143,Z 69,A -129.4656,B 24.8917,C -2.4017,E1 24.9112,E2 213.4692} C_DIS
LIN {X -31.6078,Y -51.9652,Z 69,A -126.3568,B 24.8923,C -2.3959,E1 24.9185,E2 210.3643} C_DIS
LIN {X -29.293,Y -53.3054,Z 69,A -123.6738,B 24.8923,C -2.3958,E1 24.9251,E2 207.6738} C_DIS
LIN {X -26.6861,Y -54.6573,Z 69,A -120.9521,B 24.8927,C -2.3915,E1 24.9319,E2 204.955} C_DIS
LIN {X -23.8336,Y -55.9593,Z 69,A -118.1485,B 24.8932,C -2.3853,E1 24.939,E2 202.1595} C_DIS
LIN {X -21.8065,Y -56.7802,Z 69,A -115.8965,B 24.8931,C -2.3873,E1 24.9449,E2 199.8979} C_DIS
LIN {X -19.3373,Y -57.6673,Z 69,A -113.2483,B 24.8929,C -2.389,E1 24.9519,E2 197.2406} C_DIS
LIN {X -15.8641,Y -58.7177,Z 69,A -110,B 24.8934,C -2.3832,E1 24.9606,E2 194.0008} C_DIS
LIN {X -11.9295,Y -59.6424,Z 69,A -106.5997,B 24.8943,C -2.3728,E1 24.9698,E2 190.6208} C_DIS
LIN {X -9.4809,Y -60.0798,Z 69,A -103.9703,B 24.8939,C -2.3782,E1 24.9771,E2 187.9762} C_DIS
LIN {X -6.6391,Y -60.4603,Z 69,A -100.9158,B 24.8932,C -2.3854,E1 24.9856,E2 184.9026} C_DIS
LIN {X -3.1454,Y -60.742,Z 69,A -97.8797,B 24.8937,C -2.3797,E1 24.9941,E2 181.8789} C_DIS
LIN {X -0.0736,Y -60.8237,Z 69,A -95.3706,B 24.8944,C -2.3719,E1 25.001,E2 179.3882} C_DIS
LIN {X -0.0736,Y -60.8237,Z 69,A -95.3706,B 24.8944,C -2.3719,E1 25.001,E2 179.3882} C_DIS
Enddeposition()
LIN {X 0.3366,Y -59.8276,Z 69,A -93.7992,B 24.8906,C -2.4147,E1 25.0057,E2 177.7154} C_DIS
Startdeposition()
$VEL.CP = VEL_PRINT
LIN {X -0.7699,Y -59.8308,Z 69,A -97.073,B 24.8949,C -2.367,E1 24.9962,E2 181.1021} C_DIS
LIN {X -5.6206,Y -59.5704,Z 69,A -101.2549,B 24.894,C -2.3766,E1 24.9846,E2 185.2626} C_DIS
LIN {X -8.4974,Y -59.2285,Z 69,A -104.7375,B 24.8953,C -2.3626,E1 24.9749,E2 188.7811} C_DIS
LIN {X -11.7867,Y -58.663,Z 69,A -107.3268,B 24.8941,C -2.376,E1 24.9679,E2 191.3412} C_DIS
LIN {X -14.1529,Y -58.137,Z 69,A -110.0049,B 24.8946,C -2.3699,E1 24.9605,E2 194.0372} C_DIS
LIN {X -16.8643,Y -57.4086,Z 69,A -112.813,B 24.8946,C -2.3693,E1 24.953,E2 196.8514} C_DIS
LIN {X -19.4847,Y -56.5745,Z 69,A -115.9368,B 24.8953,C -2.3617,E1 24.9446,E2 199.9992} C_DIS
LIN {X -23.0102,Y -55.2341,Z 69,A -118.9643,B 24.894,C -2.3766,E1 24.9369,E2 202.9979} C_DIS
LIN {X -25.7288,Y -54.0211,Z 69,A -121.8285,B 24.8938,C -2.3795,E1 24.9296,E2 205.8622} C_DIS
LIN {X -29.0937,Y -52.2855,Z 69,A -125.0205,B 24.8926,C -2.3925,E1 24.9218,E2 209.0321} C_DIS
LIN {X -32.3125,Y -50.3598,Z 69,A -128.776,B 24.8924,C -2.3945,E1 24.9128,E2 212.7944} C_DIS
LIN {X -34.3647,Y -48.9831,Z 69,A -131.6995,B 24.893,C -2.3877,E1 24.906,E2 215.7439} C_DIS
LIN {X -36.3256,Y -47.5471,Z 69,A -133.7334,B 24.8922,C -2.3973,E1 24.9015,E2 217.7624} C_DIS
LIN {X -38.5018,Y -45.8033,Z 69,A -136.4266,B 24.8918,C -2.4017,E1 24.8957,E2 220.4553} C_DIS
LIN {X -40.9867,Y -43.5924,Z 69,A -139.5929,B 24.8912,C -2.4083,E1 24.8892,E2 223.6186} C_DIS
LIN {X -42.949,Y -41.661,Z 69,A -142.2661,B 24.8907,C -2.4131,E1 24.8839,E2 226.2917} C_DIS
LIN {X -44.8712,Y -39.5838,Z 69,A -145.1929,B 24.8905,C -2.4151,E1 24.8784,E2 229.2268} C_DIS
LIN {X -47.2705,Y -36.6845,Z 69,A -148.1557,B 24.8887,C -2.4351,E1 24.8733,E2 232.1555} C_DIS
LIN {X -48.5123,Y -35.0269,Z 69,A -150.5911,B 24.889,C -2.4316,E1 24.8692,E2 234.611} C_DIS
LIN {X -50.1158,Y -32.6911,Z 69,A -153.9042,B 24.8894,C -2.4277,E1 24.864,E2 237.9501} C_DIS
LIN {X -52.1394,Y -29.3554,Z 69,A -157.0859,B 24.8876,C -2.4473,E1 24.8596,E2 241.1014} C_DIS
LIN {X -53.6714,Y -26.4502,Z 69,A -160.3575,B 24.887,C -2.4536,E1 24.8554,E2 244.3755} C_DIS
LIN {X -55.4598,Y -22.4597,Z 69,A -164.3417,B 24.8856,C -2.4689,E1 24.851,E2 248.345} C_DIS
LIN {X -56.3654,Y -20.0807,Z 69,A -166.9288,B 24.8852,C -2.4733,E1 24.8485,E2 250.9363} C_DIS
LIN {X -57.5399,Y -16.4129,Z 69,A -170.7354,B 24.8844,C -2.4822,E1 24.8454,E2 254.7438} C_DIS
LIN {X -58.2013,Y -13.8891,Z 69,A -173.187,B 24.8836,C -2.4905,E1 24.8437,E2 257.1898} C_DIS
LIN {X -58.8189,Y -10.9845,Z 69,A -175.9885,B 24.8827,C -2.4999,E1 24.8422,E2 259.9854} C_DIS
LIN {X -59.303,Y -7.9656,Z 69,A -179.0319,B 24.882,C -2.5069,E1 24.841,E2 263.0301} C_DIS
LIN {X -59.5401,Y -5.9388,Z 69,A 179.0253,B 24.8814,C -2.5132,E1 24.8404,E2 264.9696} C_DIS
LIN {X -59.7636,Y -2.9418,Z 69,A 176.1242,B 24.8806,C -2.5218,E1 24.8399,E2 267.8675} C_DIS
LIN {X -59.8354,Y 0.2924,Z 69,A 172.8244,B 24.88,C -2.5281,E1 24.8399,E2 271.1722} C_DIS
LIN {X -59.7216,Y 3.6832,Z 69,A 169.5032,B 24.8792,C -2.5371,E1 24.8403,E2 274.4918} C_DIS
LIN {X -59.3499,Y 7.6032,Z 69,A 165.4638,B 24.8785,C -2.5444,E1 24.8415,E2 278.5379} C_DIS
LIN {X -58.7283,Y 11.455,Z 69,A 162.1284,B 24.8767,C -2.563,E1 24.8432,E2 281.8486} C_DIS
LIN {X -57.7634,Y 15.6076,Z 69,A 158.3013,B 24.875,C -2.5801,E1 24.8457,E2 285.6573} C_DIS
LIN {X -57.0371,Y 18.0862,Z 69,A 155.5661,B 24.8747,C -2.5832,E1 24.8479,E2 288.4009} C_DIS
LIN {X -56.0976,Y 20.8179,Z 69,A 152.8025,B 24.8739,C -2.5916,E1 24.8505,E2 291.16} C_DIS
LIN {X -54.4886,Y 24.723,Z 69,A 148.6739,B 24.8729,C -2.6022,E1 24.855,E2 295.2861} C_DIS
LIN {X -53.1046,Y 27.5724,Z 69,A 145.5189,B 24.8722,C -2.6089,E1 24.859,E2 298.4421} C_DIS
LIN {X -51.0461,Y 31.2176,Z 69,A 141.0585,B 24.8719,C -2.6124,E1 24.8653,E2 302.9172} C_DIS
LIN {X -48.7013,Y 34.762,Z 69,A 137.2325,B 24.8704,C -2.6276,E1 24.8714,E2 306.7257} C_DIS
LIN {X -46.2647,Y 37.9462,Z 69,A 133.58,B 24.869,C -2.6409,E1 24.8777,E2 310.3637} C_DIS
LIN {X -43.8785,Y 40.6815,Z 69,A 130.1714,B 24.8681,C -2.6507,E1 24.884,E2 313.7641} C_DIS
LIN {X -41.8776,Y 42.738,Z 69,A 127.0337,B 24.8681,C -2.6502,E1 24.8902,E2 316.9162} C_DIS
LIN {X -39.2174,Y 45.1912,Z 69,A 123.7144,B 24.8671,C -2.6606,E1 24.8971,E2 320.2239} C_DIS
LIN {X -35.8979,Y 47.8702,Z 69,A 120.222,B 24.8651,C -2.68,E1 24.9047,E2 323.6829} C_DIS
LIN {X -34.1788,Y 49.1124,Z 69,A 117.0337,B 24.8668,C -2.6629,E1 24.9121,E2 326.923} C_DIS
LIN {X -31.2111,Y 51.05,Z 69,A 113.214,B 24.867,C -2.6613,E1 24.9213,E2 330.7583} C_DIS
LIN {X -27.7219,Y 53.0259,Z 69,A 110.5829,B 24.8641,C -2.6899,E1 24.9276,E2 333.3286} C_DIS
LIN {X -24.5829,Y 54.5518,Z 69,A 107.4201,B 24.8633,C -2.6984,E1 24.9355,E2 336.4791} C_DIS
LIN {X -22.192,Y 55.5682,Z 69,A 104.2142,B 24.8643,C -2.6882,E1 24.9439,E2 339.7165} C_DIS
LIN {X -18.8795,Y 56.7789,Z 69,A 101.3263,B 24.8629,C -2.7016,E1 24.9514,E2 342.578} C_DIS
LIN {X -16.2487,Y 57.5864,Z 69,A 98.7147,B 24.8626,C -2.705,E1 24.9584,E2 345.186} C_DIS
LIN {X -11.5994,Y 58.7005,Z 69,A 94.4621,B 24.8615,C -2.7154,E1 24.97,E2 349.4194} C_DIS
LIN {X -8.1368,Y 59.2793,Z 69,A 90.792,B 24.8619,C -2.7116,E1 24.9801,E2 353.1017} C_DIS
LIN {X -5.0266,Y 59.6234,Z 69,A 87.3925,B 24.8626,C -2.7052,E1 24.9896,E2 356.5186} C_DIS
LIN {X 0.2568,Y 59.8344,Z 69,A 82.0763,B 24.8629,C -2.7014,E1 25.0044,E2 361.844} C_DIS
LIN {X 3.8048,Y 59.7142,Z 69,A 78.4108,B 24.8635,C -2.6961,E1 25.0147,E2 365.5207} C_DIS
LIN {X 7.0193,Y 59.4218,Z 69,A 75.6493,B 24.8629,C -2.7023,E1 25.0223,E2 368.2655} C_DIS
LIN {X 10.6642,Y 58.8769,Z 69,A 72.6268,B 24.8619,C -2.7116,E1 25.0306,E2 371.2629} C_DIS
LIN {X 13.8298,Y 58.2152,Z 69,A 69.479,B 24.8622,C -2.709,E1 25.0392,E2 374.4126} C_DIS
LIN {X 16.2316,Y 57.5913,Z 69,A 66.5491,B 24.8635,C -2.6958,E1 25.0471,E2 377.369} C_DIS
LIN {X 20.1123,Y 56.3543,Z 69,A 63.23,B 24.8626,C -2.7049,E1 25.0558,E2 380.6601} C_DIS
LIN {X 22.9476,Y 55.2605,Z 69,A 60.4059,B 24.8627,C -2.7039,E1 25.0631,E2 383.4804} C_DIS
LIN {X 26.221,Y 53.7846,Z 69,A 56.9123,B 24.8632,C -2.6987,E1 25.072,E2 386.9773} C_DIS
LIN {X 29.7351,Y 51.9234,Z 69,A 53.7015,B 24.8624,C -2.7067,E1 25.0798,E2 390.1598} C_DIS
LIN {X 32.7271,Y 50.092,Z 69,A 49.8725,B 24.864,C -2.6914,E1 25.089,E2 394.0131} C_DIS
LIN {X 34.9148,Y 48.5923,Z 69,A 47.2565,B 24.8646,C -2.6855,E1 25.0949,E2 396.634} C_DIS
LIN {X 37.1635,Y 46.8945,Z 69,A 44.5772,B 24.865,C -2.6811,E1 25.1009,E2 399.3138} C_DIS
LIN {X 38.9309,Y 45.4381,Z 69,A 42.7112,B 24.8647,C -2.6843,E1 25.1048,E2 401.165} C_DIS
LIN {X 41.5939,Y 43.0136,Z 69,A 38.9285,B 24.8661,C -2.6699,E1 25.1126,E2 404.9665} C_DIS
LIN {X 43.6665,Y 40.908,Z 69,A 36.1158,B 24.8667,C -2.6643,E1 25.1181,E2 407.7805} C_DIS
LIN {X 46.4012,Y 37.7778,Z 69,A 32.1735,B 24.8675,C -2.6561,E1 25.1252,E2 411.7241} C_DIS
LIN {X 48.1655,Y 35.5012,Z 69,A 29.4009,B 24.8682,C -2.6492,E1 25.1299,E2 414.5} C_DIS
LIN {X 50.0856,Y 32.7369,Z 69,A 26.3397,B 24.8687,C -2.6448,E1 25.1347,E2 417.5563} C_DIS
LIN {X 51.8651,Y 29.8366,Z 69,A 23.1839,B 24.8693,C -2.6388,E1 25.1392,E2 420.7102} C_DIS
LIN {X 53.1094,Y 27.5633,Z 69,A 19.9913,B 24.8716,C -2.6156,E1 25.1434,E2 423.9409} C_DIS
LIN {X 54.567,Y 24.549,Z 69,A 17.376,B 24.8711,C -2.6204,E1 25.1465,E2 426.5306} C_DIS
LIN {X 55.5969,Y 22.1194,Z 69,A 14.8748,B 24.8717,C -2.6138,E1 25.1491,E2 429.0335} C_DIS
LIN {X 56.5766,Y 19.4781,Z 69,A 12.1386,B 24.8726,C -2.6051,E1 25.1517,E2 431.7751} C_DIS
LIN {X 57.3616,Y 17.0253,Z 69,A 9.6697,B 24.8733,C -2.5978,E1 25.1537,E2 434.2473} C_DIS
LIN {X 58.3409,Y 13.2886,Z 69,A 5.7044,B 24.875,C -2.5803,E1 25.1564,E2 438.2309} C_DIS
LIN {X 59.0421,Y 9.7094,Z 69,A 2.3373,B 24.8758,C -2.5726,E1 25.1581,E2 441.5966} C_DIS
LIN {X 59.5549,Y 5.778,Z 69,A -0.7731,B 24.8753,C -2.5771,E1 25.1591,E2 444.6779} C_DIS
LIN {X 59.7751,Y 2.6761,Z 69,A -4.4917,B 24.8779,C -2.5501,E1 25.1597,E2 448.4382} C_DIS
LIN {X 59.834,Y -0.4719,Z 69,A -7.21,B 24.8782,C -2.5476,E1 25.1597,E2 451.1462} C_DIS
LIN {X 59.7432,Y -3.3114,Z 69,A -9.9293,B 24.879,C -2.5391,E1 25.1594,E2 453.8696} C_DIS
LIN {X 59.5571,Y -5.7648,Z 69,A -12.127,B 24.8793,C -2.5354,E1 25.1589,E2 456.063} C_DIS
LIN {X 59.1462,Y -9.0528,Z 69,A -14.9339,B 24.8795,C -2.5341,E1 25.1579,E2 458.8563} C_DIS
LIN {X 58.8778,Y -10.6595,Z 69,A -17.012,B 24.8811,C -2.5168,E1 25.1568,E2 460.9631} C_DIS
LIN {X 58.2273,Y -13.7802,Z 69,A -19.8321,B 24.8815,C -2.5128,E1 25.1551,E2 463.7763} C_DIS
LIN {X 57.6716,Y -15.9444,Z 69,A -22.3374,B 24.8829,C -2.4975,E1 25.1533,E2 466.3034} C_DIS
LIN {X 56.8519,Y -18.6586,Z 69,A -24.7476,B 24.883,C -2.4963,E1 25.1513,E2 468.7027} C_DIS
LIN {X 55.8561,Y -21.4565,Z 69,A -27.8524,B 24.8844,C -2.4815,E1 25.1482,E2 471.8251} C_DIS
LIN {X 54.1877,Y -25.3758,Z 69,A -31.3678,B 24.8844,C -2.4827,E1 25.1443,E2 475.3185} C_DIS
LIN {X 52.5271,Y -28.6547,Z 69,A -35.4444,B 24.8865,C -2.4593,E1 25.139,E2 479.4288} C_DIS
LIN {X 50.9884,Y -31.3126,Z 69,A -37.9155,B 24.8862,C -2.4621,E1 25.1355,E2 481.8808} C_DIS
LIN {X 48.8001,Y -34.6234,Z 69,A -41.3373,B 24.8864,C -2.4606,E1 25.1302,E2 485.2892} C_DIS
LIN {X 47.7246,Y -36.0917,Z 69,A -44.4358,B 24.8897,C -2.4243,E1 25.1249,E2 488.4587} C_DIS
LIN {X 45.6472,Y -38.6856,Z 69,A -46.2311,B 24.8875,C -2.4483,E1 25.1218,E2 490.1889} C_DIS
LIN {X 43.8551,Y -40.707,Z 69,A -49.7329,B 24.89,C -2.4206,E1 25.1152,E2 493.7407} C_DIS
LIN {X 41.1664,Y -43.4235,Z 69,A -53.9434,B 24.892,C -2.3994,E1 25.1066,E2 497.9839} C_DIS
LIN {X 38.4654,Y -45.8335,Z 69,A -57.0127,B 24.8918,C -2.4007,E1 25.1001,E2 501.0382} C_DIS
LIN {X 34.2708,Y -49.0484,Z 69,A -61.4085,B 24.8914,C -2.4054,E1 25.0903,E2 505.4072} C_DIS
LIN {X 31.9886,Y -50.5672,Z 69,A -64.1325,B 24.8921,C -2.3982,E1 25.0839,E2 508.1394} C_DIS
LIN {X 29.9404,Y -51.8055,Z 69,A -66.679,B 24.893,C -2.3884,E1 25.0777,E2 510.7015} C_DIS
LIN {X 25.8988,Y -53.9395,Z 69,A -70.3494,B 24.8922,C -2.397,E1 25.0687,E2 514.3413} C_DIS
LIN {X 24.3097,Y -54.6748,Z 69,A -73.1893,B 24.8947,C -2.3687,E1 25.0613,E2 517.2412} C_DIS
LIN {X 21.3396,Y -55.9004,Z 69,A -75.2913,B 24.8932,C -2.3859,E1 25.0559,E2 519.2978} C_DIS
LIN {X 19.0996,Y -56.7047,Z 69,A -77.9877,B 24.8942,C -2.3739,E1 25.0487,E2 522.0172} C_DIS
LIN {X 15.8792,Y -57.6901,Z 69,A -80.8879,B 24.8939,C -2.3774,E1 25.041,E2 524.9042} C_DIS
LIN {X 12.8765,Y -58.4331,Z 69,A -83.9274,B 24.8943,C -2.373,E1 25.0327,E2 527.9501} C_DIS
LIN {X 9.8603,Y -59.0168,Z 69,A -86.6373,B 24.8941,C -2.3756,E1 25.0253,E2 530.6506} C_DIS
LIN {X 8.1276,Y -59.281,Z 69,A -88.9853,B 24.8955,C -2.3602,E1 25.0187,E2 533.033} C_DIS
LIN {X 4.4309,Y -59.6716,Z 69,A -91.7237,B 24.8941,C -2.3758,E1 25.0112,E2 535.733} C_DIS
LIN {X 0.3366,Y -59.8276,Z 69,A -93.798,B 24.8906,C -2.4142,E1 25.0058,E2 537.7154} C_DIS
Enddeposition()
LIN {X 0.3366,Y -59.8276,Z 69,A -93.798,B 24.8906,C -2.4142,E1 25.0058,E2 537.7154} C_DIS
Startdeposition()
$VEL.CP = VEL_PRINT
LIN {X 2.1764,Y -58.8062,Z 69,A -92.6455,B 24.8903,C -2.4176,E1 25.0089,E2 536.5551} C_DIS
LIN {X 5.5613,Y -58.5836,Z 69,A -89.5329,B 24.8905,C -2.4151,E1 25.0176,E2 533.4499} C_DIS
LIN {X 8.5406,Y -58.2243,Z 69,A -86.7205,B 24.8905,C -2.4147,E1 25.0253,E2 530.6411} C_DIS
LIN {X 11.1043,Y -57.7896,Z 69,A -84.0639,B 24.8901,C -2.4194,E1 25.0327,E2 527.9762} C_DIS
LIN {X 14.7085,Y -56.979,Z 69,A -80.5458,B 24.89,C -2.4211,E1 25.0422,E2 524.459} C_DIS
LIN {X 17.149,Y -56.2933,Z 69,A -77.5084,B 24.8886,C -2.4364,E1 25.0504,E2 521.3906} C_DIS
LIN {X 21.074,Y -54.9445,Z 69,A -73.412,B 24.888,C -2.443,E1 25.0612,E2 517.2873} C_DIS
LIN {X 24.9732,Y -53.2851,Z 69,A -69.6559,B 24.8882,C -2.4408,E1 25.0707,E2 513.5456} C_DIS
LIN {X 28.0747,Y -51.718,Z 69,A -66.6381,B 24.8884,C -2.4382,E1 25.0781,E2 510.5425} C_DIS
LIN {X 30.3916,Y -50.391,Z 69,A -63.7702,B 24.8874,C -2.449,E1 25.085,E2 507.6578} C_DIS
LIN {X 33.3174,Y -48.5078,Z 69,A -60.9813,B 24.8881,C -2.4419,E1 25.0915,E2 504.8951} C_DIS
LIN {X 35.0829,Y -47.2458,Z 69,A -58.4595,B 24.8868,C -2.4556,E1 25.0972,E2 502.3498} C_DIS
LIN {X 37.6672,Y -45.2121,Z 69,A -55.354,B 24.8864,C -2.4603,E1 25.104,E2 499.2449} C_DIS
LIN {X 40.853,Y -42.3553,Z 69,A -51.456,B 24.8861,C -2.4636,E1 25.112,E2 495.3548} C_DIS
LIN {X 42.7708,Y -40.418,Z 69,A -48.4251,B 24.8847,C -2.4788,E1 25.1179,E2 492.3009} C_DIS
LIN {X 44.8242,Y -38.1279,Z 69,A -45.379,B 24.8839,C -2.4876,E1 25.1235,E2 489.2478} C_DIS
LIN {X 47.4357,Y -34.8253,Z 69,A -41.7033,B 24.8838,C -2.4884,E1 25.1297,E2 485.5875} C_DIS
LIN {X 49.1182,Y -32.409,Z 69,A -38.5864,B 24.8825,C -2.5022,E1 25.1347,E2 482.4535} C_DIS
LIN {X 50.746,Y -29.7962,Z 69,A -35.7368,B 24.882,C -2.5071,E1 25.1388,E2 479.6067} C_DIS
LIN {X 52.0011,Y -27.5471,Z 69,A -32.837,B 24.8804,C -2.5237,E1 25.1426,E2 476.683} C_DIS
LIN {X 53.5907,Y -24.3105,Z 69,A -29.5856,B 24.8801,C -2.5278,E1 25.1465,E2 473.4393} C_DIS
LIN {X 54.8115,Y -21.4163,Z 69,A -26.277,B 24.8786,C -2.543,E1 25.15,E2 470.1131} C_DIS
LIN {X 56.1281,Y -17.6819,Z 69,A -22.0651,B 24.8766,C -2.5634,E1 25.1536,E2 465.8768} C_DIS
LIN {X 57.2593,Y -13.5805,Z 69,A -18.5362,B 24.8768,C -2.5615,E1 25.156,E2 462.3728} C_DIS
LIN {X 58.0889,Y -9.4183,Z 69,A -14.613,B 24.8761,C -2.5695,E1 25.158,E2 458.4537} C_DIS
LIN {X 58.4831,Y -6.535,Z 69,A -11.816,B 24.8753,C -2.5776,E1 25.159,E2 455.6541} C_DIS
LIN {X 58.7326,Y -3.6678,Z 69,A -8.8698,B 24.8741,C -2.5899,E1 25.1596,E2 452.6963} C_DIS
LIN {X 58.8449,Y -0.5685,Z 69,A -6.1295,B 24.8738,C -2.5927,E1 25.1598,E2 449.9656} C_DIS
LIN {X 58.7848,Y 2.7064,Z 69,A -2.4892,B 24.8717,C -2.6136,E1 25.1594,E2 446.2976} C_DIS
LIN {X 58.5622,Y 5.7883,Z 69,A 0.2557,B 24.8714,C -2.6166,E1 25.1588,E2 443.5618} C_DIS
LIN {X 58.1768,Y 8.8558,Z 69,A 3.0831,B 24.871,C -2.6216,E1 25.1577,E2 440.7392} C_DIS
LIN {X 57.7197,Y 11.4666,Z 69,A 5.8713,B 24.8697,C -2.6344,E1 25.1562,E2 437.937} C_DIS
LIN {X 56.7901,Y 15.4219,Z 69,A 9.6384,B 24.8689,C -2.6419,E1 25.1537,E2 434.1742} C_DIS
LIN {X 56.2473,Y 17.2975,Z 69,A 11.8546,B 24.8676,C -2.655,E1 25.1519,E2 431.9396} C_DIS
LIN {X 54.9456,Y 21.0709,Z 69,A 15.3934,B 24.8673,C -2.658,E1 25.1485,E2 428.4135} C_DIS
LIN {X 53.8403,Y 23.7535,Z 69,A 17.8956,B 24.8673,C -2.6584,E1 25.1458,E2 425.9241} C_DIS
LIN {X 51.9094,Y 27.7214,Z 69,A 22.1205,B 24.8663,C -2.6684,E1 25.1406,E2 421.698} C_DIS
LIN {X 49.9738,Y 31.0737,Z 69,A 26.2758,B 24.8644,C -2.6872,E1 25.1346,E2 417.5195} C_DIS
LIN {X 47.6034,Y 34.5962,Z 69,A 30.3046,B 24.8636,C -2.695,E1 25.1282,E2 413.492} C_DIS
LIN {X 45.9229,Y 36.7986,Z 69,A 33.3999,B 24.862,C -2.7105,E1 25.1228,E2 410.3746} C_DIS
LIN {X 43.399,Y 39.7426,Z 69,A 36.6798,B 24.8623,C -2.7076,E1 25.1168,E2 407.1163} C_DIS
LIN {X 41.4355,Y 41.7859,Z 69,A 39.2439,B 24.8622,C -2.709,E1 25.1118,E2 404.5599} C_DIS
LIN {X 39.2092,Y 43.8815,Z 69,A 42.4082,B 24.8611,C -2.7191,E1 25.1053,E2 401.3843} C_DIS
LIN {X 36.8996,Y 45.8411,Z 69,A 45.415,B 24.8604,C -2.7259,E1 25.0988,E2 398.373} C_DIS
LIN {X 34.5757,Y 47.6185,Z 69,A 48.2071,B 24.8601,C -2.7295,E1 25.0926,E2 395.5823} C_DIS
LIN {X 33.0584,Y 48.6836,Z 69,A 50.5364,B 24.8586,C -2.7441,E1 25.0871,E2 393.2263} C_DIS
LIN {X 29.4882,Y 50.9257,Z 69,A 53.6502,B 24.8602,C -2.7283,E1 25.0798,E2 390.1598} C_DIS
LIN {X 25.9955,Y 52.794,Z 69,A 57.26,B 24.8602,C -2.728,E1 25.071,E2 386.5611} C_DIS
LIN {X 23.1452,Y 54.1049,Z 69,A 61.0906,B 24.8582,C -2.7481,E1 25.0611,E2 382.6923} C_DIS
LIN {X 20.4726,Y 55.1718,Z 69,A 63.7926,B 24.8582,C -2.7486,E1 25.0541,E2 379.995} C_DIS
LIN {X 17.3735,Y 56.2237,Z 69,A 67.3702,B 24.857,C -2.7594,E1 25.0445,E2 376.3983} C_DIS
LIN {X 14.5606,Y 57.017,Z 69,A 69.7767,B 24.8578,C -2.7519,E1 25.0381,E2 374.0135} C_DIS
LIN {X 11.8546,Y 57.6404,Z 69,A 72.52,B 24.8575,C -2.754,E1 25.0306,E2 371.2688} C_DIS
LIN {X 9.8007,Y 58.025,Z 69,A 75.5915,B 24.8552,C -2.7764,E1 25.022,E2 368.1471} C_DIS
LIN {X 6.2198,Y 58.5172,Z 69,A 78.2013,B 24.8571,C -2.758,E1 25.0149,E2 365.5829} C_DIS
LIN {X 3.592,Y 58.7376,Z 69,A 80.4017,B 24.8579,C -2.7506,E1 25.0088,E2 363.4013} C_DIS
LIN {X 0.4743,Y 58.845,Z 69,A 84.1556,B 24.8564,C -2.7648,E1 24.9982,E2 359.6142} C_DIS
LIN {X -3.0147,Y 58.77,Z 69,A 86.8956,B 24.8579,C -2.7505,E1 24.9907,E2 356.9078} C_DIS
LIN {X -5.4173,Y 58.5969,Z 69,A 89.422,B 24.8576,C -2.753,E1 24.9836,E2 354.3742} C_DIS
LIN {X -7.6724,Y 58.3446,Z 69,A 91.4427,B 24.8582,C -2.748,E1 24.978,E2 352.364} C_DIS
LIN {X -10.8925,Y 57.8304,Z 69,A 94.4,B 24.8588,C -2.7415,E1 24.9699,E2 349.4195} C_DIS
LIN {X -13.2699,Y 57.3311,Z 69,A 97.4664,B 24.8576,C -2.7531,E1 24.9615,E2 346.3214} C_DIS
LIN {X -16.6413,Y 56.4448,Z 69,A 100.6147,B 24.8585,C -2.7448,E1 24.9531,E2 343.188} C_DIS
LIN {X -19.3795,Y 55.5643,Z 69,A 103.5998,B 24.8585,C -2.7451,E1 24.9451,E2 340.1968} C_DIS
LIN {X -22.7121,Y 54.2874,Z 69,A 106.6784,B 24.8597,C -2.7328,E1 24.9372,E2 337.1406} C_DIS
LIN {X -25.7655,Y 52.9068,Z 69,A 110.4438,B 24.8593,C -2.7374,E1 24.9276,E2 333.3548} C_DIS
LIN {X -30.459,Y 50.3508,Z 69,A 115.2259,B 24.861,C -2.7206,E1 24.9161,E2 328.5989} C_DIS
LIN {X -32.8058,Y 48.8546,Z 69,A 118.313,B 24.8608,C -2.7224,E1 24.9088,E2 325.4973} C_DIS
LIN {X -35.1498,Y 47.1962,Z 69,A 121.3167,B 24.861,C -2.7206,E1 24.902,E2 322.4873} C_DIS
LIN {X -38.8368,Y 44.2117,Z 69,A 126.0122,B 24.8619,C -2.712,E1 24.892,E2 317.7944} C_DIS
LIN {X -42.4399,Y 40.7652,Z 69,A 130.8895,B 24.863,C -2.7009,E1 24.8824,E2 312.923} C_DIS
LIN {X -45.6256,Y 37.1654,Z 69,A 135.625,B 24.8641,C -2.69,E1 24.8738,E2 308.1917} C_DIS
LIN {X -48.3099,Y 33.602,Z 69,A 139.2473,B 24.8666,C -2.6656,E1 24.8679,E2 304.6102} C_DIS
LIN {X -49.3508,Y 32.0554,Z 69,A 141.5274,B 24.8662,C -2.6688,E1 24.8644,E2 302.311} C_DIS
LIN {X -51.0729,Y 29.2321,Z 69,A 145.0463,B 24.8666,C -2.6651,E1 24.8594,E2 298.7828} C_DIS
LIN {X -52.8402,Y 25.9022,Z 69,A 148.6933,B 24.8677,C -2.654,E1 24.8549,E2 295.1427} C_DIS
LIN {X -54.2006,Y 22.9183,Z 69,A 151.3055,B 24.8697,C -2.6344,E1 24.852,E2 292.5631} C_DIS
LIN {X -55.6512,Y 19.1313,Z 69,A 155.5329,B 24.8704,C -2.6272,E1 24.8479,E2 288.3289} C_DIS
LIN {X -56.3018,Y 17.1216,Z 69,A 157.916,B 24.8704,C -2.6266,E1 24.8459,E2 285.9335} C_DIS
LIN {X -57.3512,Y 13.1829,Z 69,A 161.2946,B 24.8727,C -2.6041,E1 24.8436,E2 282.5892} C_DIS
LIN {X -57.8608,Y 10.7316,Z 69,A 163.893,B 24.8732,C -2.5992,E1 24.8422,E2 279.987} C_DIS
LIN {X -58.5143,Y 6.248,Z 69,A 168.5142,B 24.8742,C -2.5889,E1 24.8405,E2 275.3628} C_DIS
LIN {X -58.7454,Y 3.4585,Z 69,A 171.0641,B 24.8753,C -2.5773,E1 24.84,E2 272.8255} C_DIS
LIN {X -58.8383,Y 1.0029,Z 69,A 173.6264,B 24.8757,C -2.5727,E1 24.8398,E2 270.2587} C_DIS
LIN {X -58.8134,Y -1.9917,Z 69,A 176.5662,B 24.8766,C -2.5639,E1 24.84,E2 267.3222} C_DIS
LIN {X -58.6558,Y -4.737,Z 69,A 178.9409,B 24.8779,C -2.5503,E1 24.8404,E2 264.9658} C_DIS
LIN {X -58.3295,Y -7.789,Z 69,A -177.2211,B 24.8774,C -2.5558,E1 24.8417,E2 261.0915} C_DIS
LIN {X -57.7026,Y -11.5515,Z 69,A -173.9837,B 24.8793,C -2.5361,E1 24.8433,E2 257.8822} C_DIS
LIN {X -57.1481,Y -14.0372,Z 69,A -171.525,B 24.88,C -2.5282,E1 24.8449,E2 255.4278} C_DIS
LIN {X -56.5232,Y -16.3764,Z 69,A -169.0445,B 24.8805,C -2.5234,E1 24.8468,E2 252.9445} C_DIS
LIN {X -55.4164,Y -19.801,Z 69,A -165.5541,B 24.8815,C -2.5129,E1 24.8499,E2 249.4592} C_DIS
LIN {X -54.702,Y -21.6948,Z 69,A -163.5951,B 24.882,C -2.5071,E1 24.8519,E2 247.5032} C_DIS
LIN {X -53.171,Y -25.2165,Z 69,A -159.9523,B 24.8832,C -2.4949,E1 24.856,E2 243.8694} C_DIS
LIN {X -51.8562,Y -27.82,Z 69,A -157.1959,B 24.884,C -2.4858,E1 24.8596,E2 241.1202} C_DIS
LIN {X -50.4512,Y -30.2938,Z 69,A -154.0302,B 24.884,C -2.4856,E1 24.864,E2 237.9383} C_DIS
LIN {X -48.1073,Y -33.8932,Z 69,A -149.9454,B 24.8852,C -2.4734,E1 24.8704,E2 233.8623} C_DIS
LIN {X -45.3058,Y -37.5543,Z 69,A -145.0677,B 24.8855,C -2.4701,E1 24.8789,E2 228.9697} C_DIS
LIN {X -42.8699,Y -40.3127,Z 69,A -141.8839,B 24.8869,C -2.4549,E1 24.8848,E2 225.8081} C_DIS
LIN {X -40.2989,Y -42.8829,Z 69,A -137.7406,B 24.8865,C -2.459,E1 24.8932,E2 221.6378} C_DIS
LIN {X -37.2417,Y -45.5638,Z 69,A -134.4848,B 24.8884,C -2.4383,E1 24.9001,E2 218.4188} C_DIS
LIN {X -33.8972,Y -48.1043,Z 69,A -130.0686,B 24.8884,C -2.4376,E1 24.91,E2 213.9887} C_DIS
LIN {X -31.6149,Y -49.6335,Z 69,A -126.7423,B 24.8877,C -2.4461,E1 24.9179,E2 210.6312} C_DIS
LIN {X -27.9753,Y -51.7719,Z 69,A -123.0847,B 24.889,C -2.4318,E1 24.9268,E2 206.9973} C_DIS
LIN {X -24.8806,Y -53.3283,Z 69,A -120.0297,B 24.8899,C -2.4216,E1 24.9344,E2 203.9586} C_DIS
LIN {X -22.3526,Y -54.4365,Z 69,A -116.1717,B 24.8881,C -2.4423,E1 24.9445,E2 200.0427} C_DIS
LIN {X -18.6182,Y -55.8242,Z 69,A -113.7729,B 24.8911,C -2.4093,E1 24.9507,E2 197.7177} C_DIS
LIN {X -16.4647,Y -56.4967,Z 69,A -111.3662,B 24.8908,C -2.412,E1 24.9571,E2 195.3005} C_DIS
LIN {X -14.0798,Y -57.1377,Z 69,A -108.8863,B 24.8908,C -2.4122,E1 24.9638,E2 192.8166} C_DIS
LIN {X -11.6438,Y -57.6836,Z 69,A -106.1422,B 24.8903,C -2.4176,E1 24.9714,E2 190.0565} C_DIS
LIN {X -8.4299,Y -58.24,Z 69,A -103.3165,B 24.891,C -2.4095,E1 24.9791,E2 187.2474} C_DIS
LIN {X -5.9055,Y -58.5501,Z 69,A -100.1867,B 24.8898,C -2.4228,E1 24.9879,E2 184.0841} C_DIS
LIN {X -0.2085,Y -58.8466,Z 69,A -94.7661,B 24.89,C -2.4207,E1 25.003,E2 178.6678} C_DIS
LIN {X -0.2085,Y -58.8466,Z 69,A -94.7661,B 24.89,C -2.4207,E1 25.003,E2 178.6678} C_DIS
Enddeposition()
LIN {X 0.3119,Y -57.8571,Z 69,A -95.2667,B 24.8904,C -2.4168,E1 25.0016,E2 179.1777} C_DIS
Startdeposition()
$VEL.CP = VEL_PRINT
LIN {X -3.4849,Y -57.7538,Z 69,A -100.208,B 24.8926,C -2.3925,E1 24.9877,E2 184.1774} C_DIS
LIN {X -6.7607,Y -57.4623,Z 69,A -103.0481,B 24.8918,C -2.4011,E1 24.9798,E2 186.9988} C_DIS
LIN {X -8.7707,Y -57.1901,Z 69,A -105.7479,B 24.893,C -2.3881,E1 24.9723,E2 189.7319} C_DIS
LIN {X -12.9694,Y -56.3863,Z 69,A -109.6777,B 24.8923,C -2.3958,E1 24.9616,E2 193.6481} C_DIS
LIN {X -17.0085,Y -55.3024,Z 69,A -113.0677,B 24.8907,C -2.4129,E1 24.9526,E2 197.0028} C_DIS
LIN {X -20.1827,Y -54.2254,Z 69,A -117.4116,B 24.8923,C -2.3962,E1 24.941,E2 201.395} C_DIS
LIN {X -23.4974,Y -52.8733,Z 69,A -120.3622,B 24.8909,C -2.411,E1 24.9335,E2 204.3172} C_DIS
LIN {X -26.2719,Y -51.5501,Z 69,A -123.5696,B 24.8909,C -2.4116,E1 24.9254,E2 207.5317} C_DIS
LIN {X -28.6656,Y -50.2588,Z 69,A -126.6915,B 24.8912,C -2.4073,E1 24.9178,E2 210.6727} C_DIS
LIN {X -31.6105,Y -48.4611,Z 69,A -129.9363,B 24.8905,C -2.4156,E1 24.9102,E2 213.9083} C_DIS
LIN {X -35.0355,Y -46.0454,Z 69,A -134.0887,B 24.8899,C -2.4226,E1 24.9008,E2 218.0587} C_DIS
LIN {X -38.4656,Y -43.2209,Z 69,A -138.2169,B 24.8887,C -2.4357,E1 24.8921,E2 222.1716} C_DIS
LIN {X -40.4924,Y -41.3274,Z 69,A -140.9883,B 24.8882,C -2.4408,E1 24.8865,E2 224.9423} C_DIS
LIN {X -42.6529,Y -39.0942,Z 69,A -144.7059,B 24.8886,C -2.4362,E1 24.8794,E2 228.6871} C_DIS
LIN {X -45.1858,Y -36.1378,Z 69,A -147.7422,B 24.8865,C -2.4593,E1 24.8741,E2 231.6824} C_DIS
LIN {X -46.6308,Y -34.252,Z 69,A -149.9904,B 24.8858,C -2.4667,E1 24.8703,E2 233.9236} C_DIS
LIN {X -48.8174,Y -31.057,Z 69,A -153.9666,B 24.8851,C -2.4738,E1 24.8641,E2 237.9027} C_DIS
LIN {X -50.6935,Y -27.8911,Z 69,A -157.416,B 24.8839,C -2.4867,E1 24.8593,E2 241.3393} C_DIS
LIN {X -51.6722,Y -26.0322,Z 69,A -159.6391,B 24.8836,C -2.4898,E1 24.8564,E2 243.5667} C_DIS
LIN {X -52.4247,Y -24.4802,Z 69,A -161.6905,B 24.8837,C -2.4887,E1 24.854,E2 245.6319} C_DIS
LIN {X -53.9546,Y -20.8951,Z 69,A -166.1495,B 24.8837,C -2.4897,E1 24.8493,E2 250.1136} C_DIS
LIN {X -55.5036,Y -16.3397,Z 69,A -170.2613,B 24.8813,C -2.5145,E1 24.8458,E2 254.1895} C_DIS
LIN {X -56.3304,Y -13.2115,Z 69,A -173.2699,B 24.8801,C -2.5274,E1 24.8437,E2 257.1849} C_DIS
LIN {X -56.8147,Y -10.9412,Z 69,A -176.0426,B 24.8801,C -2.5266,E1 24.8422,E2 259.976} C_DIS
LIN {X -57.356,Y -7.6124,Z 69,A -179.1623,B 24.8788,C -2.5405,E1 24.8409,E2 263.081} C_DIS
LIN {X -57.681,Y -4.5312,Z 69,A 178.3318,B 24.877,C -2.5594,E1 24.8403,E2 265.5567} C_DIS
LIN {X -57.7949,Y -2.7262,Z 69,A 175.9413,B 24.8774,C -2.555,E1 24.8399,E2 267.9719} C_DIS
LIN {X -57.8542,Y 0.7539,Z 69,A 172.2679,B 24.8768,C -2.5622,E1 24.8399,E2 271.6505} C_DIS
LIN {X -57.7385,Y 3.725,Z 69,A 169.5397,B 24.8755,C -2.575,E1 24.8402,E2 274.3644} C_DIS
LIN {X -57.5667,Y 5.8091,Z 69,A 167.2321,B 24.8753,C -2.5777,E1 24.8409,E2 276.6795} C_DIS
LIN {X -57.0702,Y 9.5195,Z 69,A 163.932,B 24.8735,C -2.596,E1 24.8422,E2 279.9553} C_DIS
LIN {X -56.5831,Y 12.0836,Z 69,A 161.1766,B 24.873,C -2.6013,E1 24.8437,E2 282.7144} C_DIS
LIN {X -55.89,Y 14.9648,Z 69,A 157.8785,B 24.8726,C -2.6044,E1 24.846,E2 286.0244} C_DIS
LIN {X -55.0802,Y 17.7147,Z 69,A 155.4584,B 24.8711,C -2.62,E1 24.8479,E2 288.421} C_DIS
LIN {X -54.1872,Y 20.2837,Z 69,A 152.4319,B 24.8708,C -2.6227,E1 24.8508,E2 291.4583} C_DIS
LIN {X -53.0889,Y 23.0046,Z 69,A 148.8725,B 24.8711,C -2.6206,E1 24.8547,E2 295.0425} C_DIS
LIN {X -51.3422,Y 26.6778,Z 69,A 144.7676,B 24.87,C -2.631,E1 24.8599,E2 299.1446} C_DIS
LIN {X -49.1166,Y 30.581,Z 69,A 140.8524,B 24.8679,C -2.6523,E1 24.8655,E2 303.0289} C_DIS
LIN {X -47.2388,Y 33.4084,Z 69,A 137.532,B 24.8669,C -2.6621,E1 24.8707,E2 306.3423} C_DIS
LIN {X -45.0208,Y 36.3424,Z 69,A 134.2698,B 24.8653,C -2.6781,E1 24.8763,E2 309.5819} C_DIS
LIN {X -43.3124,Y 38.3634,Z 69,A 131.2991,B 24.8653,C -2.6787,E1 24.8817,E2 312.5646} C_DIS
LIN {X -41.6843,Y 40.1253,Z 69,A 129.3221,B 24.864,C -2.6913,E1 24.8855,E2 314.5201} C_DIS
LIN {X -39.9374,Y 41.8654,Z 69,A 126.3701,B 24.8643,C -2.6882,E1 24.8914,E2 317.4918} C_DIS
LIN {X -38.018,Y 43.6149,Z 69,A 123.7052,B 24.8639,C -2.6923,E1 24.897,E2 320.1574} C_DIS
LIN {X -34.9483,Y 46.1112,Z 69,A 120.1906,B 24.8623,C -2.7076,E1 24.9046,E2 323.6485} C_DIS
LIN {X -32.8751,Y 47.6118,Z 69,A 117.1891,B 24.8626,C -2.7044,E1 24.9115,E2 326.668} C_DIS
LIN {X -30.4216,Y 49.2161,Z 69,A 114.8531,B 24.8611,C -2.7198,E1 24.917,E2 328.9746} C_DIS
LIN {X -27.3183,Y 51.0042,Z 69,A 110.4355,B 24.862,C -2.7103,E1 24.9278,E2 333.4276} C_DIS
LIN {X -24.1622,Y 52.5727,Z 69,A 107.7606,B 24.86,C -2.7304,E1 24.9345,E2 336.0616} C_DIS
LIN {X -20.7507,Y 54.0103,Z 69,A 103.8134,B 24.86,C -2.7303,E1 24.9447,E2 340.018} C_DIS
LIN {X -18.123,Y 54.9481,Z 69,A 100.3251,B 24.861,C -2.7203,E1 24.954,E2 343.5365} C_DIS
LIN {X -14.2694,Y 56.0716,Z 69,A 96.2411,B 24.8608,C -2.7222,E1 24.965,E2 347.622} C_DIS
LIN {X -11.1398,Y 56.7765,Z 69,A 94.381,B 24.858,C -2.7495,E1 24.9699,E2 349.4194} C_DIS
LIN {X -7.6603,Y 57.3492,Z 69,A 90.5986,B 24.8583,C -2.7463,E1 24.9804,E2 353.2128} C_DIS
LIN {X -5.0277,Y 57.6405,Z 69,A 87.5752,B 24.859,C -2.74,E1 24.9888,E2 356.2529} C_DIS
LIN {X -2.1267,Y 57.8202,Z 69,A 85.0614,B 24.8582,C -2.748,E1 24.9958,E2 358.7482} C_DIS
LIN {X 0.733,Y 57.855,Z 69,A 81.8506,B 24.8589,C -2.7412,E1 25.0048,E2 361.9751} C_DIS
LIN {X 3.6969,Y 57.7402,Z 69,A 78.9712,B 24.8587,C -2.7424,E1 25.0128,E2 364.8506} C_DIS
LIN {X 7.8082,Y 57.3303,Z 69,A 74.6205,B 24.8593,C -2.7366,E1 25.0249,E2 369.2119} C_DIS
LIN {X 11.3027,Y 56.745,Z 69,A 71.4509,B 24.8588,C -2.742,E1 25.0336,E2 372.365} C_DIS
LIN {X 13.782,Y 56.1933,Z 69,A 69.1605,B 24.8585,C -2.7452,E1 25.0398,E2 374.6446} C_DIS
LIN {X 17.2643,Y 55.2231,Z 69,A 65.0189,B 24.8599,C -2.7313,E1 25.0509,E2 378.8121} C_DIS
LIN {X 20.703,Y 54.0284,Z 69,A 61.8462,B 24.8593,C -2.7369,E1 25.0592,E2 381.9649} C_DIS
LIN {X 24.0018,Y 52.6452,Z 69,A 58.5237,B 24.8593,C -2.7377,E1 25.0677,E2 385.2775} C_DIS
LIN {X 25.7813,Y 51.7973,Z 69,A 55.6668,B 24.8614,C -2.7165,E1 25.075,E2 388.1771} C_DIS
LIN {X 28.7226,Y 50.226,Z 69,A 52.7382,B 24.8611,C -2.7198,E1 25.0821,E2 391.0893} C_DIS
LIN {X 31.9064,Y 48.2661,Z 69,A 49.2145,B 24.8613,C -2.7179,E1 25.0903,E2 394.6061} C_DIS
LIN {X 34.3799,Y 46.5372,Z 69,A 46.3955,B 24.8614,C -2.7165,E1 25.0967,E2 397.4185} C_DIS
LIN {X 37.5188,Y 44.045,Z 69,A 42.2154,B 24.8626,C -2.7046,E1 25.1058,E2 401.6108} C_DIS
LIN {X 40.3545,Y 41.4634,Z 69,A 38.6456,B 24.8629,C -2.7019,E1 25.113,E2 405.1723} C_DIS
LIN {X 42.3483,Y 39.4241,Z 69,A 35.8829,B 24.8634,C -2.6973,E1 25.1183,E2 407.9342} C_DIS
LIN {X 44.3061,Y 37.2103,Z 69,A 33.0216,B 24.8639,C -2.6921,E1 25.1236,E2 410.7947} C_DIS
LIN {X 46.0145,Y 35.0768,Z 69,A 29.8709,B 24.8655,C -2.6759,E1 25.129,E2 413.969} C_DIS
LIN {X 48.1617,Y 32.0645,Z 69,A 26.3421,B 24.8662,C -2.6698,E1 25.1346,E2 417.4948} C_DIS
LIN {X 50.906,Y 27.4993,Z 69,A 21.4732,B 24.8666,C -2.6651,E1 25.1414,E2 422.3498} C_DIS
LIN {X 52.7488,Y 23.7737,Z 69,A 17.3101,B 24.8679,C -2.6527,E1 25.1465,E2 426.5198} C_DIS
LIN {X 53.8474,Y 21.1681,Z 69,A 14.1861,B 24.8694,C -2.6374,E1 25.1497,E2 429.6628} C_DIS
LIN {X 55.5077,Y 16.3261,Z 69,A 9.4447,B 24.8701,C -2.63,E1 25.1538,E2 434.3949} C_DIS
LIN {X 56.3592,Y 13.0871,Z 69,A 6.1604,B 24.871,C -2.6207,E1 25.1561,E2 437.6821} C_DIS
LIN {X 56.9987,Y 9.9412,Z 69,A 2.732,B 24.8726,C -2.6053,E1 25.1579,E2 441.127} C_DIS
LIN {X 57.4739,Y 6.6614,Z 69,A -0.0612,B 24.8725,C -2.6063,E1 25.1589,E2 443.9011} C_DIS
LIN {X 57.667,Y 4.707,Z 69,A -2.623,B 24.8744,C -2.5861,E1 25.1595,E2 446.4956} C_DIS
LIN {X 57.8599,Y -0.1144,Z 69,A -6.994,B 24.875,C -2.5804,E1 25.1598,E2 450.8541} C_DIS
LIN {X 57.7613,Y -3.359,Z 69,A -10.1802,B 24.8759,C -2.5709,E1 25.1594,E2 454.0438} C_DIS
LIN {X 57.5465,Y -6.0019,Z 69,A -12.5531,B 24.8762,C -2.5684,E1 25.1588,E2 456.4084} C_DIS
LIN {X 57.2738,Y -8.2059,Z 69,A -14.6856,B 24.8767,C -2.563,E1 25.158,E2 458.5411} C_DIS
LIN {X 56.8033,Y -11.0006,Z 69,A -18.1593,B 24.879,C -2.5388,E1 25.1562,E2 462.0516} C_DIS
LIN {X 55.705,Y -15.6398,Z 69,A -22.6047,B 24.8798,C -2.5305,E1 25.1532,E2 466.4912} C_DIS
LIN {X 54.765,Y -18.6669,Z 69,A -26.1974,B 24.8817,C -2.5105,E1 25.15,E2 470.1108} C_DIS
LIN {X 53.3209,Y -22.4612,Z 69,A -29.8122,B 24.882,C -2.5076,E1 25.1462,E2 473.7124} C_DIS
LIN {X 51.9791,Y -25.4146,Z 69,A -32.9797,B 24.8828,C -2.4992,E1 25.1424,E2 476.8828} C_DIS
LIN {X 50.0142,Y -29.0911,Z 69,A -36.7305,B 24.8831,C -2.496,E1 25.1373,E2 480.6217} C_DIS
LIN {X 47.7705,Y -32.6436,Z 69,A -40.6331,B 24.8836,C -2.4903,E1 25.1315,E2 484.518} C_DIS
LIN {X 46.3269,Y -34.662,Z 69,A -43.5804,B 24.8852,C -2.4726,E1 25.1266,E2 487.493} C_DIS
LIN {X 44.1189,Y -37.4321,Z 69,A -46.7973,B 24.8855,C -2.4701,E1 25.1209,E2 490.701} C_DIS
LIN {X 42.3308,Y -39.4427,Z 69,A -49.9071,B 24.887,C -2.4535,E1 25.115,E2 493.8363} C_DIS
LIN {X 40.5048,Y -41.3163,Z 69,A -52.4106,B 24.8874,C -2.4493,E1 25.11,E2 496.3393} C_DIS
LIN {X 37.9403,Y -43.6827,Z 69,A -55.4759,B 24.8874,C -2.4501,E1 25.1036,E2 499.3904} C_DIS
LIN {X 35.6394,Y -45.5801,Z 69,A -58.6825,B 24.8884,C -2.4381,E1 25.0966,E2 502.6132} C_DIS
LIN {X 32.928,Y -47.575,Z 69,A -61.4965,B 24.888,C -2.4428,E1 25.0903,E2 505.4062} C_DIS
LIN {X 29.4287,Y -49.8154,Z 69,A -65.6166,B 24.8887,C -2.435,E1 25.0806,E2 509.5316} C_DIS
LIN {X 26.625,Y -51.3695,Z 69,A -69.3515,B 24.8903,C -2.4175,E1 25.0713,E2 513.2975} C_DIS
LIN {X 23.7196,Y -52.7732,Z 69,A -72.541,B 24.8908,C -2.4127,E1 25.0632,E2 516.4901} C_DIS
LIN {X 20.8083,Y -53.9885,Z 69,A -74.9981,B 24.8899,C -2.4226,E1 25.0569,E2 518.9182} C_DIS
LIN {X 16.8843,Y -55.3409,Z 69,A -79.0616,B 24.8902,C -2.4185,E1 25.0462,E2 522.9834} C_DIS
LIN {X 15.1024,Y -55.8529,Z 69,A -81.8358,B 24.8922,C -2.3969,E1 25.0386,E2 525.8045} C_DIS
LIN {X 10.1774,Y -56.9566,Z 69,A -86.4701,B 24.8919,C -2.4002,E1 25.0259,E2 530.4253} C_DIS
LIN {X 7.273,Y -57.4,Z 69,A -89.0605,B 24.8915,C -2.4048,E1 25.0188,E2 533.0025} C_DIS
LIN {X 5.0279,Y -57.6405,Z 69,A -91.2623,B 24.8915,C -2.4043,E1 25.0127,E2 535.2041} C_DIS
LIN {X 2.4842,Y -57.8053,Z 69,A -94.054,B 24.8921,C -2.3979,E1 25.0049,E2 538.01} C_DIS
LIN {X 0.3119,Y -57.8571,Z 69,A -95.2659,B 24.8904,C -2.4164,E1 25.0016,E2 539.1777} C_DIS
Enddeposition()
LIN {X 0.3119,Y -57.8571,Z 69,A -95.2659,B 24.8904,C -2.4164,E1 25.0016,E2 539.1777} C_DIS
Startdeposition()
$VEL.CP = VEL_PRINT
LIN {X 1.8241,Y -56.8414,Z 69,A -92.9781,B 24.8874,C -2.4495,E1 25.0082,E2 536.8119} C_DIS
LIN {X 5.0902,Y -56.6424,Z 69,A -89.8448,B 24.8876,C -2.4477,E1 25.0169,E2 533.6844} C_DIS
LIN {X 8.1314,Y -56.2864,Z 69,A -86.7241,B 24.8873,C -2.4504,E1 25.0256,E2 530.5599} C_DIS
LIN {X 11.7236,Y -55.6498,Z 69,A -83.545,B 24.888,C -2.443,E1 25.0342,E2 527.4019} C_DIS
LIN {X 13.7452,Y -55.1843,Z 69,A -80.8383,B 24.8866,C -2.458,E1 25.0417,E2 524.6635} C_DIS
LIN {X 16.6196,Y -54.3885,Z 69,A -77.172,B 24.885,C -2.4756,E1 25.0516,E2 520.962} C_DIS
LIN {X 19.8209,Y -53.3052,Z 69,A -75.0123,B 24.8871,C -2.4532,E1 25.0571,E2 518.8599} C_DIS
LIN {X 22.9235,Y -52.0463,Z 69,A -71.5986,B 24.8865,C -2.4588,E1 25.0659,E2 515.4408} C_DIS
LIN {X 24.5744,Y -51.2871,Z 69,A -69.4018,B 24.8855,C -2.4696,E1 25.0715,E2 513.2241} C_DIS
LIN {X 27.7593,Y -49.6355,Z 69,A -66.2344,B 24.8859,C -2.4659,E1 25.0792,E2 510.0743} C_DIS
LIN {X 30.2067,Y -48.1853,Z 69,A -62.5665,B 24.8837,C -2.4888,E1 25.0881,E2 506.3637} C_DIS
LIN {X 32.9094,Y -46.3816,Z 69,A -59.3909,B 24.8833,C -2.4932,E1 25.0953,E2 503.1888} C_DIS
LIN {X 36.2534,Y -43.8174,Z 69,A -55.3746,B 24.883,C -2.4971,E1 25.1041,E2 499.1782} C_DIS
LIN {X 39.2569,Y -41.1488,Z 69,A -51.7047,B 24.8829,C -2.4979,E1 25.1116,E2 495.5212} C_DIS
LIN {X 40.7136,Y -39.7086,Z 69,A -49.1361,B 24.8813,C -2.5143,E1 25.1167,E2 492.9248} C_DIS
LIN {X 43.4136,Y -36.7363,Z 69,A -45.2572,B 24.8807,C -2.5207,E1 25.1238,E2 489.0482} C_DIS
LIN {X 45.9301,Y -33.5363,Z 69,A -41.5512,B 24.8806,C -2.5225,E1 25.1301,E2 485.3555} C_DIS
LIN {X 47.8496,Y -30.7356,Z 69,A -37.7399,B 24.8788,C -2.5409,E1 25.136,E2 481.5198} C_DIS
LIN {X 49.3023,Y -28.3468,Z 69,A -35.0232,B 24.8783,C -2.5466,E1 25.1399,E2 478.8036} C_DIS
LIN {X 50.9731,Y -25.2191,Z 69,A -31.939,B 24.8783,C -2.5457,E1 25.1438,E2 475.7377} C_DIS
LIN {X 51.7515,Y -23.5817,Z 69,A -29.3158,B 24.8761,C -2.5695,E1 25.1469,E2 473.0725} C_DIS
LIN {X 53.0384,Y -20.5248,Z 69,A -25.8821,B 24.8749,C -2.5817,E1 25.1504,E2 469.629} C_DIS
LIN {X 54.1821,Y -17.2805,Z 69,A -22.3675,B 24.8737,C -2.5935,E1 25.1535,E2 466.1065} C_DIS
LIN {X 55.3227,Y -13.1817,Z 69,A -19.1745,B 24.8749,C -2.5814,E1 25.1557,E2 462.9605} C_DIS
LIN {X 55.8608,Y -10.6696,Z 69,A -16.1627,B 24.8732,C -2.5993,E1 25.1574,E2 459.9239} C_DIS
LIN {X 56.3515,Y -7.6687,Z 69,A -13.1296,B 24.8723,C -2.6082,E1 25.1586,E2 456.8874} C_DIS
LIN {X 56.6731,Y -4.7402,Z 69,A -9.9085,B 24.8708,C -2.6235,E1 25.1595,E2 453.6493} C_DIS
LIN {X 56.8592,Y -1.1426,Z 69,A -6.9757,B 24.8712,C -2.6188,E1 25.1598,E2 450.7451} C_DIS
LIN {X 56.8669,Y 0.6823,Z 69,A -4.5756,B 24.8694,C -2.6376,E1 25.1598,E2 448.3149} C_DIS
LIN {X 56.6914,Y 4.5101,Z 69,A -1.1054,B 24.8691,C -2.6407,E1 25.1591,E2 444.858} C_DIS
LIN {X 56.3532,Y 7.658,Z 69,A 2.6026,B 24.8669,C -2.6626,E1 25.1578,E2 441.1201} C_DIS
LIN {X 55.6031,Y 11.9402,Z 69,A 6.3106,B 24.8671,C -2.6604,E1 25.1559,E2 437.4388} C_DIS
LIN {X 54.9665,Y 14.5946,Z 69,A 9.113,B 24.8661,C -2.6699,E1 25.154,E2 434.6303} C_DIS
LIN {X 54.4352,Y 16.4666,Z 69,A 11.2125,B 24.8652,C -2.6789,E1 25.1523,E2 432.5214} C_DIS
LIN {X 53.5667,Y 19.1038,Z 69,A 14.5362,B 24.8632,C -2.6991,E1 25.1493,E2 429.1686} C_DIS
LIN {X 52.0062,Y 23.0154,Z 69,A 18.4246,B 24.8628,C -2.703,E1 25.145,E2 425.2924} C_DIS
LIN {X 50.3667,Y 26.4096,Z 69,A 21.752,B 24.8628,C -2.7027,E1 25.1409,E2 421.9835} C_DIS
LIN {X 48.4692,Y 29.7499,Z 69,A 25.7948,B 24.8614,C -2.7167,E1 25.1352,E2 417.9284} C_DIS
LIN {X 47.198,Y 31.7276,Z 69,A 28.4528,B 24.8601,C -2.7291,E1 25.1311,E2 415.2541} C_DIS
LIN {X 44.5229,Y 35.3836,Z 69,A 32.5637,B 24.8601,C -2.7299,E1 25.1242,E2 411.161} C_DIS
LIN {X 42.6065,Y 37.6689,Z 69,A 35.5975,B 24.8593,C -2.7374,E1 25.1187,E2 408.1233} C_DIS
LIN {X 40.8507,Y 39.5664,Z 69,A 38.2889,B 24.8585,C -2.7449,E1 25.1135,E2 405.4258} C_DIS
LIN {X 38.7327,Y 41.6429,Z 69,A 41.2679,B 24.8579,C -2.7507,E1 25.1075,E2 402.4453} C_DIS
LIN {X 36.8127,Y 43.3485,Z 69,A 43.8991,B 24.8573,C -2.7566,E1 25.1019,E2 399.8104} C_DIS
LIN {X 33.8694,Y 45.6863,Z 69,A 48.1906,B 24.8554,C -2.7742,E1 25.0924,E2 395.4929} C_DIS
LIN {X 30.1623,Y 48.213,Z 69,A 51.9499,B 24.8564,C -2.765,E1 25.0837,E2 391.768} C_DIS
LIN {X 27.8003,Y 49.6126,Z 69,A 54.9269,B 24.8555,C -2.7733,E1 25.0764,E2 388.7801} C_DIS
LIN {X 25.5671,Y 50.8002,Z 69,A 57.6279,B 24.8549,C -2.7797,E1 25.0697,E2 386.0713} C_DIS
LIN {X 22.106,Y 52.3983,Z 69,A 61.2662,B 24.8549,C -2.7797,E1 25.0604,E2 382.442} C_DIS
LIN {X 19.8093,Y 53.3101,Z 69,A 63.7643,B 24.8546,C -2.7822,E1 25.0539,E2 379.9434} C_DIS
LIN {X 17.2967,Y 54.1762,Z 69,A 66.2872,B 24.8547,C -2.7812,E1 25.0473,E2 377.4277} C_DIS
LIN {X 14.9398,Y 54.8733,Z 69,A 69.0784,B 24.8539,C -2.7893,E1 25.0397,E2 374.6219} C_DIS
LIN {X 12.2848,Y 55.5281,Z 69,A 71.6158,B 24.8542,C -2.7863,E1 25.0328,E2 372.0951} C_DIS
LIN {X 10.2913,Y 55.9321,Z 69,A 74.6161,B 24.8521,C -2.8063,E1 25.0245,E2 369.0505} C_DIS
LIN {X 6.9873,Y 56.4395,Z 69,A 76.9618,B 24.8541,C -2.7865,E1 25.0181,E2 366.7538} C_DIS
LIN {X 4.2223,Y 56.7144,Z 69,A 80.0935,B 24.8534,C -2.7933,E1 25.0094,E2 363.6077} C_DIS
LIN {X 0.969,Y 56.8624,Z 69,A 83.0669,B 24.8541,C -2.787,E1 25.0011,E2 360.6502} C_DIS
LIN {X -1.8871,Y 56.8394,Z 69,A 86.0541,B 24.854,C -2.7883,E1 24.9928,E2 357.6593} C_DIS
LIN {X -4.668,Y 56.6788,Z 69,A 89.0223,B 24.8538,C -2.7903,E1 24.9845,E2 354.6853} C_DIS
LIN {X -8.6803,Y 56.2042,Z 69,A 93.2585,B 24.8537,C -2.7909,E1 24.9728,E2 350.4443} C_DIS
LIN {X -13.335,Y 55.2849,Z 69,A 97.4302,B 24.8553,C -2.7754,E1 24.9614,E2 346.3046} C_DIS
LIN {X -15.0523,Y 54.8429,Z 69,A 99.6622,B 24.8546,C -2.7819,E1 24.9554,E2 344.0537} C_DIS
LIN {X -18.6657,Y 53.7204,Z 69,A 103.0889,B 24.8558,C -2.7704,E1 24.9463,E2 340.6483} C_DIS
LIN {X -21.4582,Y 52.6669,Z 69,A 106.5055,B 24.8555,C -2.7739,E1 24.9374,E2 337.216} C_DIS
LIN {X -24.1929,Y 51.4685,Z 69,A 110.2371,B 24.8546,C -2.7826,E1 24.9279,E2 333.4542} C_DIS
LIN {X -27.1159,Y 49.9899,Z 69,A 112.9804,B 24.8562,C -2.767,E1 24.9212,E2 330.7404} C_DIS
LIN {X -30.9513,Y 47.7111,Z 69,A 116.8145,B 24.8583,C -2.747,E1 24.9122,E2 326.9421} C_DIS
LIN {X -33.3068,Y 46.0978,Z 69,A 119.8435,B 24.8586,C -2.7441,E1 24.9052,E2 323.9097} C_DIS
LIN {X -34.7461,Y 45.0219,Z 69,A 121.953,B 24.8584,C -2.7456,E1 24.9005,E2 321.789} C_DIS
LIN {X -37.3054,Y 42.9254,Z 69,A 125.2577,B 24.8592,C -2.7378,E1 24.8935,E2 318.4901} C_DIS
Enddeposition()
END
